LIN {X 0,Y 195.393,Z 454.313,A -85,B 0,C 180,E1 -23353.111,E2 -23353.111} C_VEL
LIN {X 0,Y 194.613,Z 444.182,A -85,B 0,C 180,E1 -23355.96,E2 -23355.96} C_VEL
LIN {X 0,Y 193.145,Z 436.002,A -85,B 0,C 180,E1 -23358.369,E2 -23358.369} C_VEL
LIN {X 0,Y 190.426,Z 427.797,A -85,B 0,C 180,E1 -23361.14,E2 -23361.14} C_VEL
LIN {X 0,Y 187.179,Z 420.29,A -85,B 0,C 180,E1 -23363.977,E2 -23363.977} C_VEL
LIN {X 0,Y 183.425,Z 413.236,A -85,B 0,C 180,E1 -23367.07,E2 -23367.07} C_VEL
LIN {X 0,Y 181.652,Z 409.98,A -85,B 0,C 180,E1 -23368.592,E2 -23368.592} C_VEL
LIN {X 0,Y 179.184,Z 405.781,A -85,B 0,C 180,E1 -23370.721,E2 -23370.721} C_VEL
LIN {X 0,Y 176.213,Z 401.753,A -85,B 0,C 180,E1 -23373.34,E2 -23373.34} C_VEL
LIN {X 0,Y 175.243,Z 399.934,A -85,B 0,C 180,E1 -23374.302,E2 -23374.302} C_VEL
LIN {X 0,Y 172.386,Z 396.823,A -85,B 0,C 180,E1 -23377.054,E2 -23377.054} C_VEL
LIN {X 0,Y 171.129,Z 394.282,A -85,B 0,C 180,E1 -23378.577,E2 -23378.577} C_VEL
LIN {X 0,Y 167.914,Z 391.613,A -85,B 0,C 180,E1 -23382.335,E2 -23382.335} C_VEL
LIN {X 0,Y 166.254,Z 388.555,A -85,B 0,C 180,E1 -23385.072,E2 -23385.072} C_VEL
LIN {X 0,Y 166.146,Z 388.15,A -85,B 0,C 180,E1 -23385.457,E2 -23385.457} C_VEL
LIN {X 0,Y 166.298,Z 387.582,A -85,B 0,C 180,E1 -23390.267,E2 -23390.267} C_VEL
LIN {X 0,Y 166.273,Z 387.45,A -85,B 0,C 180,E1 -23395.15,E2 -23395.15} C_VEL
LIN {X 0,Y 166.781,Z 387.561,A -85,B 0,C 180,E1 -23400,E2 -23400} C_VEL
LIN {X 0,Y 166.489,Z 388.269,A -85,B 0,C 180,E1 -23404.843,E2 -23404.843} C_VEL
LIN {X 0,Y 166.58,Z 389.214,A -85,B 0,C 180,E1 -23409.715,E2 -23409.715} C_VEL
LIN {X 0,Y 166.697,Z 390.162,A -85,B 0,C 180,E1 -23412.858,E2 -23412.858} C_VEL
LIN {X 0,Y 168.099,Z 393.319,A -85,B 0,C 180,E1 -23415.147,E2 -23415.147} C_VEL
LIN {X 0,Y 171.251,Z 396.71,A -85,B 0,C 180,E1 -23418.855,E2 -23418.855} C_VEL
LIN {X 0,Y 171.981,Z 397.621,A -85,B 0,C 180,E1 -23419.625,E2 -23419.625} C_VEL
LIN {X 0,Y 173.741,Z 401.026,A -85,B 0,C 180,E1 -23421.583,E2 -23421.583} C_VEL
LIN {X 0,Y 176.205,Z 403.912,A -85,B 0,C 180,E1 -23423.818,E2 -23423.818} C_VEL
LIN {X 0,Y 178.445,Z 408.052,A -85,B 0,C 180,E1 -23425.903,E2 -23425.903} C_VEL
LIN {X 0,Y 179.87,Z 410.061,A -85,B 0,C 180,E1 -23427.085,E2 -23427.085} C_VEL
LIN {X 0,Y 182.312,Z 414.458,A -85,B 0,C 180,E1 -23429.122,E2 -23429.122} C_VEL
LIN {X 0,Y 183.669,Z 417.262,A -85,B 0,C 180,E1 -23430.305,E2 -23430.305} C_VEL
LIN {X 0,Y 185.712,Z 421.013,A -85,B 0,C 180,E1 -23431.912,E2 -23431.912} C_VEL
LIN {X 0,Y 189.672,Z 429.746,A -85,B 0,C 180,E1 -23435.182,E2 -23435.182} C_VEL
LIN {X 0,Y 193.411,Z 440.1,A -85,B 0,C 180,E1 -23438.605,E2 -23438.605} C_VEL
LIN {X 0,Y 195.794,Z 448.846,A -85,B 0,C 180,E1 -23441.232,E2 -23441.232} C_VEL
LIN {X 0,Y 195.872,Z 455.455,A -85,B 0,C 180,E1 -23442.769,E2 -23442.769} C_VEL
LIN {X 0,Y 194.863,Z 467.884,A -85,B 0,C 180,E1 -23445.671,E2 -23445.671} C_VEL
LIN {X 0,Y 193.774,Z 474.064,A -85,B 0,C 180,E1 -23447.152,E2 -23447.152} C_VEL
LIN {X 0,Y 188.97,Z 484.708,A -85,B 0,C 180,E1 -23449.394,E2 -23449.394} C_VEL
LIN {X 0,Y 183.723,Z 495.484,A -85,B 0,C 180,E1 -23452.261,E2 -23452.261} C_VEL
LIN {X 0,Y 179.025,Z 504.532,A -85,B 0,C 180,E1 -23455.287,E2 -23455.287} C_VEL
LIN {X 0,Y 174.37,Z 513.451,A -85,B 0,C 180,E1 -23459.076,E2 -23459.076} C_VEL
LIN {X 0,Y 170.178,Z 520.786,A -85,B 0,C 180,E1 -23462.981,E2 -23462.981} C_VEL
LIN {X 0,Y 166.593,Z 527.552,A -85,B 0,C 180,E1 -23467.686,E2 -23467.686} C_VEL
LIN {X 0,Y 164.027,Z 532.799,A -85,B 0,C 180,E1 -23472.546,E2 -23472.546} C_VEL
LIN {X 0,Y 162.495,Z 536.663,A -85,B 0,C 180,E1 -23477.511,E2 -23477.511} C_VEL
LIN {X 0,Y 161.925,Z 539.221,A -85,B 0,C 180,E1 -23482.518,E2 -23482.518} C_VEL
LIN {X 0,Y 161.964,Z 540.31,A -85,B 0,C 180,E1 -23486.392,E2 -23486.392} C_VEL
LIN {X 0,Y 162.166,Z 540.683,A -85,B 0,C 180,E1 -23490,E2 -23490} C_VEL
LIN {X 0,Y 161.945,Z 540.01,A -85,B 0,C 180,E1 -23494.979,E2 -23494.979} C_VEL
LIN {X 0,Y 162.104,Z 538.06,A -85,B 0,C 180,E1 -23499.994,E2 -23499.994} C_VEL
LIN {X 0,Y 163.129,Z 534.845,A -85,B 0,C 180,E1 -23504.981,E2 -23504.981} C_VEL
LIN {X 0,Y 165.326,Z 529.872,A -85,B 0,C 180,E1 -23510.278,E2 -23510.278} C_VEL
LIN {X 0,Y 165.698,Z 527.731,A -85,B 0,C 180,E1 -23512.183,E2 -23512.183} C_VEL
LIN {X 0,Y 164.607,Z 520.58,A -85,B 0,C 180,E1 -23517.854,E2 -23517.854} C_VEL
LIN {X 0,Y 165.371,Z 517.795,A -85,B 0,C 180,E1 -23519.642,E2 -23519.642} C_VEL
LIN {X 0,Y 165.926,Z 516.803,A -85,B 0,C 180,E1 -23520.201,E2 -23520.201} C_VEL
LIN {X 0,Y 170.168,Z 509.415,A -85,B 0,C 180,E1 -23523.835,E2 -23523.835} C_VEL
LIN {X 0,Y 175.497,Z 499.649,A -85,B 0,C 180,E1 -23527.641,E2 -23527.641} C_VEL
LIN {X 0,Y 180.783,Z 489.726,A -85,B 0,C 180,E1 -23530.629,E2 -23530.629} C_VEL
LIN {X 0,Y 185.516,Z 480.008,A -85,B 0,C 180,E1 -23532.993,E2 -23532.993} C_VEL
LIN {X 0,Y 187.889,Z 474.908,A -85,B 0,C 180,E1 -23534.042,E2 -23534.042} C_VEL
LIN {X 0,Y 189.104,Z 468.404,A -85,B 0,C 180,E1 -23535.678,E2 -23535.678} C_VEL
LIN {X 0,Y 190.178,Z 457.705,A -85,B 0,C 180,E1 -23538.304,E2 -23538.304} C_VEL
LIN {X 0,Y 190.26,Z 451.9,A -85,B 0,C 180,E1 -23539.727,E2 -23539.727} C_VEL
LIN {X 0,Y 188.045,Z 442.99,A -85,B 0,C 180,E1 -23542.603,E2 -23542.603} C_VEL
LIN {X 0,Y 184.882,Z 433.595,A -85,B 0,C 180,E1 -23545.896,E2 -23545.896} C_VEL
LIN {X 0,Y 180.855,Z 424.352,A -85,B 0,C 180,E1 -23549.657,E2 -23549.657} C_VEL
LIN {X 0,Y 178.545,Z 419.648,A -85,B 0,C 180,E1 -23551.813,E2 -23551.813} C_VEL
LIN {X 0,Y 176.166,Z 414.939,A -85,B 0,C 180,E1 -23554.13,E2 -23554.13} C_VEL
LIN {X 0,Y 173.783,Z 410.864,A -85,B 0,C 180,E1 -23556.462,E2 -23556.462} C_VEL
LIN {X 0,Y 173.009,Z 409.372,A -85,B 0,C 180,E1 -23557.3,E2 -23557.3} C_VEL
LIN {X 0,Y 170.455,Z 405.778,A -85,B 0,C 180,E1 -23560.026,E2 -23560.026} C_VEL
LIN {X 0,Y 169.384,Z 403.444,A -85,B 0,C 180,E1 -23561.4,E2 -23561.4} C_VEL
LIN {X 0,Y 166.445,Z 399.985,A -85,B 0,C 180,E1 -23565.149,E2 -23565.149} C_VEL
LIN {X 0,Y 165.014,Z 396.727,A -85,B 0,C 180,E1 -23567.705,E2 -23567.705} C_VEL
LIN {X 0,Y 161.043,Z 391.856,A -85,B 0,C 180,E1 -23579.375,E2 -23579.375} C_VEL
LIN {X 0,Y 160.969,Z 391.971,A -85,B 0,C 180,E1 -23583.129,E2 -23583.129} C_VEL
LIN {X 0,Y 162.436,Z 393.477,A -85,B 0,C 180,E1 -23589.967,E2 -23589.967} C_VEL
LIN {X 0,Y 164.736,Z 395.178,A -85,B 0,C 180,E1 -23594.668,E2 -23594.668} C_VEL
LIN {X 0,Y 166.487,Z 398.565,A -85,B 0,C 180,E1 -23597.822,E2 -23597.822} C_VEL
LIN {X 0,Y 169.25,Z 401.27,A -85,B 0,C 180,E1 -23601.306,E2 -23601.306} C_VEL
LIN {X 0,Y 171.208,Z 404.731,A -85,B 0,C 180,E1 -23603.754,E2 -23603.754} C_VEL
LIN {X 0,Y 173.066,Z 406.867,A -85,B 0,C 180,E1 -23605.642,E2 -23605.642} C_VEL
LIN {X 0,Y 175.344,Z 410.764,A -85,B 0,C 180,E1 -23608.016,E2 -23608.016} C_VEL
LIN {X 0,Y 176.352,Z 412.26,A -85,B 0,C 180,E1 -23608.977,E2 -23608.977} C_VEL
LIN {X 0,Y 178.854,Z 416.578,A -85,B 0,C 180,E1 -23611.332,E2 -23611.332} C_VEL
LIN {X 0,Y 182.86,Z 425.001,A -85,B 0,C 180,E1 -23615.206,E2 -23615.206} C_VEL
LIN {X 0,Y 185.603,Z 431.859,A -85,B 0,C 180,E1 -23617.976,E2 -23617.976} C_VEL
LIN {X 0,Y 188.024,Z 439.877,A -85,B 0,C 180,E1 -23620.855,E2 -23620.855} C_VEL
LIN {X 0,Y 189.257,Z 448.168,A -85,B 0,C 180,E1 -23623.433,E2 -23623.433} C_VEL
LIN {X 0,Y 189.561,Z 457.642,A -85,B 0,C 180,E1 -23626.248,E2 -23626.248} C_VEL
LIN {X 0,Y 189.172,Z 465.85,A -85,B 0,C 180,E1 -23628.72,E2 -23628.72} C_VEL
LIN {X 0,Y 184.394,Z 476.022,A -85,B 0,C 180,E1 -23631.032,E2 -23631.032} C_VEL
LIN {X 0,Y 179.225,Z 486.127,A -85,B 0,C 180,E1 -23633.971,E2 -23633.971} C_VEL
LIN {X 0,Y 174.332,Z 494.554,A -85,B 0,C 180,E1 -23637.027,E2 -23637.027} C_VEL
LIN {X 0,Y 169.265,Z 502.826,A -85,B 0,C 180,E1 -23640.883,E2 -23640.883} C_VEL
LIN {X 0,Y 165.213,Z 509.295,A -85,B 0,C 180,E1 -23644.825,E2 -23644.825} C_VEL
LIN {X 0,Y 162.079,Z 513.891,A -85,B 0,C 180,E1 -23648.372,E2 -23648.372} C_VEL
LIN {X 0,Y 158.968,Z 518.703,A -85,B 0,C 180,E1 -23653.3,E2 -23653.3} C_VEL
LIN {X 0,Y 157.248,Z 521.421,A -85,B 0,C 180,E1 -23657.087,E2 -23657.087} C_VEL
LIN {X 0,Y 155.856,Z 523.863,A -85,B 0,C 180,E1 -23662.225,E2 -23662.225} C_VEL
LIN {X 0,Y 155.244,Z 525.075,A -85,B 0,C 180,E1 -23667.406,E2 -23667.406} C_VEL
LIN {X 0,Y 155.243,Z 525.092,A -85,B 0,C 180,E1 -23672.595,E2 -23672.595} C_VEL
LIN {X 0,Y 155.843,Z 523.918,A -85,B 0,C 180,E1 -23677.776,E2 -23677.776} C_VEL
LIN {X 0,Y 157.224,Z 521.516,A -85,B 0,C 180,E1 -23682.915,E2 -23682.915} C_VEL
LIN {X 0,Y 159.622,Z 517.803,A -85,B 0,C 180,E1 -23687.951,E2 -23687.951} C_VEL
LIN {X 0,Y 162.96,Z 512.68,A -85,B 0,C 180,E1 -23692.84,E2 -23692.84} C_VEL
LIN {X 0,Y 167.574,Z 505.93,A -85,B 0,C 180,E1 -23697.474,E2 -23697.474} C_VEL
LIN {X 0,Y 171.316,Z 499.691,A -85,B 0,C 180,E1 -23700.851,E2 -23700.851} C_VEL
LIN {X 0,Y 175.795,Z 492.225,A -85,B 0,C 180,E1 -23704.036,E2 -23704.036} C_VEL
LIN {X 0,Y 180.803,Z 483.334,A -85,B 0,C 180,E1 -23707.05,E2 -23707.05} C_VEL
LIN {X 0,Y 185.27,Z 474.58,A -85,B 0,C 180,E1 -23709.45,E2 -23709.45} C_VEL
LIN {X 0,Y 189.178,Z 466.217,A -85,B 0,C 180,E1 -23711.332,E2 -23711.332} C_VEL
LIN {X 0,Y 189.7,Z 457.039,A -85,B 0,C 180,E1 -23714.074,E2 -23714.074} C_VEL
LIN {X 0,Y 189.241,Z 447.251,A -85,B 0,C 180,E1 -23717.016,E2 -23717.016} C_VEL
LIN {X 0,Y 188.199,Z 440.269,A -85,B 0,C 180,E1 -23719.191,E2 -23719.191} C_VEL
LIN {X 0,Y 185.8,Z 432.24,A -85,B 0,C 180,E1 -23722.072,E2 -23722.072} C_VEL
LIN {X 0,Y 183.073,Z 425.374,A -85,B 0,C 180,E1 -23724.841,E2 -23724.841} C_VEL
LIN {X 0,Y 180.248,Z 419.479,A -85,B 0,C 180,E1 -23727.532,E2 -23727.532} C_VEL
LIN {X 0,Y 177.7,Z 414.784,A -85,B 0,C 180,E1 -23729.963,E2 -23729.963} C_VEL
LIN {X 0,Y 175.829,Z 411.344,A -85,B 0,C 180,E1 -23731.825,E2 -23731.825} C_VEL
LIN {X 0,Y 173.238,Z 407.243,A -85,B 0,C 180,E1 -23734.466,E2 -23734.466} C_VEL
LIN {X 0,Y 172.591,Z 406.168,A -85,B 0,C 180,E1 -23735.169,E2 -23735.169} C_VEL
LIN {X 0,Y 169.982,Z 402.838,A -85,B 0,C 180,E1 -23738.074,E2 -23738.074} C_VEL
LIN {X 0,Y 169.081,Z 400.884,A -85,B 0,C 180,E1 -23739.31,E2 -23739.31} C_VEL
LIN {X 0,Y 166.009,Z 397.887,A -85,B 0,C 180,E1 -23743.395,E2 -23743.395} C_VEL
LIN {X 0,Y 164.617,Z 394.969,A -85,B 0,C 180,E1 -23746.124,E2 -23746.124} C_VEL
LIN {X 0,Y 161.437,Z 392.628,A -85,B 0,C 180,E1 -23755.005,E2 -23755.005} C_VEL
LIN {X 0,Y 161.292,Z 392.143,A -85,B 0,C 180,E1 -23760.312,E2 -23760.312} C_VEL
LIN {X 0,Y 165.093,Z 396.741,A -85,B 0,C 180,E1 -23771.977,E2 -23771.977} C_VEL
LIN {X 0,Y 166.773,Z 400.471,A -85,B 0,C 180,E1 -23774.997,E2 -23774.997} C_VEL
LIN {X 0,Y 169.727,Z 403.84,A -85,B 0,C 180,E1 -23778.717,E2 -23778.717} C_VEL
LIN {X 0,Y 171.482,Z 407.457,A -85,B 0,C 180,E1 -23780.919,E2 -23780.919} C_VEL
LIN {X 0,Y 173.548,Z 410.102,A -85,B 0,C 180,E1 -23783.019,E2 -23783.019} C_VEL
LIN {X 0,Y 175.603,Z 414.134,A -85,B 0,C 180,E1 -23785.165,E2 -23785.165} C_VEL
LIN {X 0,Y 176.756,Z 415.923,A -85,B 0,C 180,E1 -23786.253,E2 -23786.253} C_VEL
LIN {X 0,Y 179.11,Z 420.459,A -85,B 0,C 180,E1 -23788.489,E2 -23788.489} C_VEL
LIN {X 0,Y 183.413,Z 429.887,A -85,B 0,C 180,E1 -23792.541,E2 -23792.541} C_VEL
LIN {X 0,Y 186.483,Z 438.016,A -85,B 0,C 180,E1 -23795.588,E2 -23795.588} C_VEL
LIN {X 0,Y 189.279,Z 447.398,A -85,B 0,C 180,E1 -23798.763,E2 -23798.763} C_VEL
LIN {X 0,Y 190.487,Z 453.178,A -85,B 0,C 180,E1 -23800.562,E2 -23800.562} C_VEL
LIN {X 0,Y 189.786,Z 463.401,A -85,B 0,C 180,E1 -23802.998,E2 -23802.998} C_VEL
LIN {X 0,Y 188.374,Z 473.627,A -85,B 0,C 180,E1 -23805.611,E2 -23805.611} C_VEL
LIN {X 0,Y 187.37,Z 476.406,A -85,B 0,C 180,E1 -23806.211,E2 -23806.211} C_VEL
LIN {X 0,Y 181.684,Z 488.144,A -85,B 0,C 180,E1 -23808.882,E2 -23808.882} C_VEL
LIN {X 0,Y 176.386,Z 498.329,A -85,B 0,C 180,E1 -23811.859,E2 -23811.859} C_VEL
LIN {X 0,Y 171.648,Z 506.944,A -85,B 0,C 180,E1 -23815.024,E2 -23815.024} C_VEL
LIN {X 0,Y 166.927,Z 515.366,A -85,B 0,C 180,E1 -23818.952,E2 -23818.952} C_VEL
LIN {X 0,Y 162.73,Z 522.284,A -85,B 0,C 180,E1 -23823.033,E2 -23823.033} C_VEL
LIN {X 0,Y 159.13,Z 528.766,A -85,B 0,C 180,E1 -23828.042,E2 -23828.042} C_VEL
LIN {X 0,Y 156.681,Z 533.558,A -85,B 0,C 180,E1 -23833.048,E2 -23833.048} C_VEL
LIN {X 0,Y 155.494,Z 536.313,A -85,B 0,C 180,E1 -23836.939,E2 -23836.939} C_VEL
LIN {X 0,Y 154.843,Z 538.873,A -85,B 0,C 180,E1 -23842.174,E2 -23842.174} C_VEL
LIN {X 0,Y 154.896,Z 540.028,A -85,B 0,C 180,E1 -23846.55,E2 -23846.55} C_VEL
LIN {X 0,Y 155.067,Z 540.337,A -85,B 0,C 180,E1 -23850,E2 -23850} C_VEL
LIN {X 0,Y 154.847,Z 539.663,A -85,B 0,C 180,E1 -23855.208,E2 -23855.208} C_VEL
LIN {X 0,Y 155.061,Z 537.716,A -85,B 0,C 180,E1 -23860.445,E2 -23860.445} C_VEL
LIN {X 0,Y 156.22,Z 534.495,A -85,B 0,C 180,E1 -23865.66,E2 -23865.66} C_VEL
LIN {X 0,Y 158.378,Z 529.931,A -85,B 0,C 180,E1 -23870.793,E2 -23870.793} C_VEL
LIN {X 0,Y 161.722,Z 523.915,A -85,B 0,C 180,E1 -23875.758,E2 -23875.758} C_VEL
LIN {X 0,Y 165.926,Z 516.803,A -85,B 0,C 180,E1 -23880.201,E2 -23880.201} C_VEL
LIN {X 0,Y 166.549,Z 514.834,A -85,B 0,C 180,E1 -23881.374,E2 -23881.374} C_VEL
LIN {X 0,Y 165.825,Z 511.72,A -85,B 0,C 180,E1 -23883.429,E2 -23883.429} C_VEL
LIN {X 0,Y 165.203,Z 508.379,A -85,B 0,C 180,E1 -23885.461,E2 -23885.461} C_VEL
LIN {X 0,Y 165.957,Z 506.053,A -85,B 0,C 180,E1 -23886.552,E2 -23886.552} C_VEL
LIN {X 0,Y 171.658,Z 496.157,A -85,B 0,C 180,E1 -23890.153,E2 -23890.153} C_VEL
LIN {X 0,Y 177.275,Z 485.624,A -85,B 0,C 180,E1 -23893.147,E2 -23893.147} C_VEL
LIN {X 0,Y 181.89,Z 476.458,A -85,B 0,C 180,E1 -23895.201,E2 -23895.201} C_VEL
LIN {X 0,Y 182.827,Z 473.07,A -85,B 0,C 180,E1 -23896.05,E2 -23896.05} C_VEL
LIN {X 0,Y 184.336,Z 462.781,A -85,B 0,C 180,E1 -23898.78,E2 -23898.78} C_VEL
LIN {X 0,Y 184.912,Z 456.848,A -85,B 0,C 180,E1 -23900.262,E2 -23900.262} C_VEL
LIN {X 0,Y 184.616,Z 454.071,A -85,B 0,C 180,E1 -23901.101,E2 -23901.101} C_VEL
LIN {X 0,Y 182.464,Z 445.092,A -85,B 0,C 180,E1 -23904.244,E2 -23904.244} C_VEL
LIN {X 0,Y 179.577,Z 436.033,A -85,B 0,C 180,E1 -23907.736,E2 -23907.736} C_VEL
LIN {X 0,Y 176.174,Z 427.807,A -85,B 0,C 180,E1 -23911.399,E2 -23911.399} C_VEL
LIN {X 0,Y 173.147,Z 421.04,A -85,B 0,C 180,E1 -23914.774,E2 -23914.774} C_VEL
LIN {X 0,Y 170.899,Z 416.946,A -85,B 0,C 180,E1 -23917.244,E2 -23917.244} C_VEL
LIN {X 0,Y 170.268,Z 415.613,A -85,B 0,C 180,E1 -23918.034,E2 -23918.034} C_VEL
LIN {X 0,Y 167.786,Z 411.62,A -85,B 0,C 180,E1 -23921.058,E2 -23921.058} C_VEL
LIN {X 0,Y 166.994,Z 409.815,A -85,B 0,C 180,E1 -23922.235,E2 -23922.235} C_VEL
LIN {X 0,Y 164.212,Z 405.951,A -85,B 0,C 180,E1 -23926.386,E2 -23926.386} C_VEL
LIN {X 0,Y 163.205,Z 403.395,A -85,B 0,C 180,E1 -23928.512,E2 -23928.512} C_VEL
LIN {X 0,Y 159.915,Z 398.72,A -85,B 0,C 180,E1 -23940,E2 -23940} C_VEL
LIN {X 0,Y 160.226,Z 399.536,A -85,B 0,C 180,E1 -23946.296,E2 -23946.296} C_VEL
LIN {X 0,Y 163.048,Z 401.904,A -85,B 0,C 180,E1 -23954.032,E2 -23954.032} C_VEL
LIN {X 0,Y 164.671,Z 405.31,A -85,B 0,C 180,E1 -23957.383,E2 -23957.383} C_VEL
LIN {X 0,Y 166.989,Z 407.8,A -85,B 0,C 180,E1 -23960.639,E2 -23960.639} C_VEL
LIN {X 0,Y 168.889,Z 411.278,A -85,B 0,C 180,E1 -23963.287,E2 -23963.287} C_VEL
LIN {X 0,Y 170.284,Z 413.024,A -85,B 0,C 180,E1 -23964.879,E2 -23964.879} C_VEL
LIN {X 0,Y 171.813,Z 416.056,A -85,B 0,C 180,E1 -23966.741,E2 -23966.741} C_VEL
LIN {X 0,Y 172.951,Z 417.649,A -85,B 0,C 180,E1 -23967.936,E2 -23967.936} C_VEL
LIN {X 0,Y 176.446,Z 424.882,A -85,B 0,C 180,E1 -23971.855,E2 -23971.855} C_VEL
LIN {X 0,Y 179.315,Z 431.782,A -85,B 0,C 180,E1 -23975.086,E2 -23975.086} C_VEL
LIN {X 0,Y 181.477,Z 437.95,A -85,B 0,C 180,E1 -23977.689,E2 -23977.689} C_VEL
LIN {X 0,Y 183.036,Z 444.155,A -85,B 0,C 180,E1 -23980.027,E2 -23980.027} C_VEL
LIN {X 0,Y 183.88,Z 452.358,A -85,B 0,C 180,E1 -23982.725,E2 -23982.725} C_VEL
LIN {X 0,Y 183.857,Z 460.777,A -85,B 0,C 180,E1 -23985.373,E2 -23985.373} C_VEL
LIN {X 0,Y 183.416,Z 467.29,A -85,B 0,C 180,E1 -23987.482,E2 -23987.482} C_VEL
LIN {X 0,Y 178.018,Z 478.189,A -85,B 0,C 180,E1 -23990.093,E2 -23990.093} C_VEL
LIN {X 0,Y 172.671,Z 487.974,A -85,B 0,C 180,E1 -23993.105,E2 -23993.105} C_VEL
LIN {X 0,Y 166.851,Z 497.382,A -85,B 0,C 180,E1 -23996.799,E2 -23996.799} C_VEL
LIN {X 0,Y 162.071,Z 504.783,A -85,B 0,C 180,E1 -24000.612,E2 -24000.612} C_VEL
LIN {X 0,Y 157.645,Z 511.263,A -85,B 0,C 180,E1 -24004.943,E2 -24004.943} C_VEL
LIN {X 0,Y 153.708,Z 516.83,A -85,B 0,C 180,E1 -24009.945,E2 -24009.945} C_VEL
LIN {X 0,Y 151.502,Z 520.061,A -85,B 0,C 180,E1 -24013.839,E2 -24013.839} C_VEL
LIN {X 0,Y 149.468,Z 523.144,A -85,B 0,C 180,E1 -24019.159,E2 -24019.159} C_VEL
LIN {X 0,Y 148.385,Z 524.966,A -85,B 0,C 180,E1 -24024.565,E2 -24024.565} C_VEL
LIN {X 0,Y 148.085,Z 525.577,A -85,B 0,C 180,E1 -24030,E2 -24030} C_VEL
LIN {X 0,Y 148.385,Z 525.001,A -85,B 0,C 180,E1 -24035.436,E2 -24035.436} C_VEL
LIN {X 0,Y 149.45,Z 523.219,A -85,B 0,C 180,E1 -24040.842,E2 -24040.842} C_VEL
LIN {X 0,Y 151.465,Z 520.173,A -85,B 0,C 180,E1 -24046.165,E2 -24046.165} C_VEL
LIN {X 0,Y 154.499,Z 515.775,A -85,B 0,C 180,E1 -24051.341,E2 -24051.341} C_VEL
LIN {X 0,Y 158.783,Z 509.873,A -85,B 0,C 180,E1 -24056.271,E2 -24056.271} C_VEL
LIN {X 0,Y 162.567,Z 504.115,A -85,B 0,C 180,E1 -24059.958,E2 -24059.958} C_VEL
LIN {X 0,Y 167.524,Z 496.479,A -85,B 0,C 180,E1 -24063.771,E2 -24063.771} C_VEL
LIN {X 0,Y 172.615,Z 488.342,A -85,B 0,C 180,E1 -24066.91,E2 -24066.91} C_VEL
LIN {X 0,Y 177.926,Z 478.632,A -85,B 0,C 180,E1 -24069.932,E2 -24069.932} C_VEL
LIN {X 0,Y 182.91,Z 468.797,A -85,B 0,C 180,E1 -24072.318,E2 -24072.318} C_VEL
LIN {X 0,Y 183.566,Z 466.653,A -85,B 0,C 180,E1 -24072.892,E2 -24072.892} C_VEL
LIN {X 0,Y 184.057,Z 457.45,A -85,B 0,C 180,E1 -24075.826,E2 -24075.826} C_VEL
LIN {X 0,Y 183.728,Z 448.637,A -85,B 0,C 180,E1 -24078.65,E2 -24078.65} C_VEL
LIN {X 0,Y 182.849,Z 442.842,A -85,B 0,C 180,E1 -24080.638,E2 -24080.638} C_VEL
LIN {X 0,Y 180.741,Z 435.478,A -85,B 0,C 180,E1 -24083.54,E2 -24083.54} C_VEL
LIN {X 0,Y 178.209,Z 428.792,A -85,B 0,C 180,E1 -24086.487,E2 -24086.487} C_VEL
LIN {X 0,Y 175.157,Z 421.928,A -85,B 0,C 180,E1 -24089.897,E2 -24089.897} C_VEL
LIN {X 0,Y 173.111,Z 417.951,A -85,B 0,C 180,E1 -24092.168,E2 -24092.168} C_VEL
LIN {X 0,Y 170.339,Z 413.123,A -85,B 0,C 180,E1 -24095.375,E2 -24095.375} C_VEL
LIN {X 0,Y 167.411,Z 408.739,A -85,B 0,C 180,E1 -24099.094,E2 -24099.094} C_VEL
LIN {X 0,Y 166.845,Z 407.464,A -85,B 0,C 180,E1 -24099.986,E2 -24099.986} C_VEL
LIN {X 0,Y 164.018,Z 404.24,A -85,B 0,C 180,E1 -24104.306,E2 -24104.306} C_VEL
LIN {X 0,Y 163.037,Z 401.815,A -85,B 0,C 180,E1 -24106.602,E2 -24106.602} C_VEL
LIN {X 0,Y 160.286,Z 399.656,A -85,B 0,C 180,E1 -24114.969,E2 -24114.969} C_VEL
LIN {X 0,Y 160.167,Z 399.081,A -85,B 0,C 180,E1 -24120,E2 -24120} C_VEL
LIN {X 0,Y 163.29,Z 403.434,A -85,B 0,C 180,E1 -24131.167,E2 -24131.167} C_VEL
LIN {X 0,Y 165.384,Z 407.876,A -85,B 0,C 180,E1 -24135.244,E2 -24135.244} C_VEL
LIN {X 0,Y 167.415,Z 410.422,A -85,B 0,C 180,E1 -24138.035,E2 -24138.035} C_VEL
LIN {X 0,Y 169.322,Z 414.314,A -85,B 0,C 180,E1 -24140.659,E2 -24140.659} C_VEL
LIN {X 0,Y 170.8,Z 416.547,A -85,B 0,C 180,E1 -24142.371,E2 -24142.371} C_VEL
LIN {X 0,Y 172.204,Z 419.621,A -85,B 0,C 180,E1 -24144.086,E2 -24144.086} C_VEL
LIN {X 0,Y 173.325,Z 421.24,A -85,B 0,C 180,E1 -24145.198,E2 -24145.198} C_VEL
LIN {X 0,Y 177.362,Z 430.35,A -85,B 0,C 180,E1 -24149.689,E2 -24149.689} C_VEL
LIN {X 0,Y 180.392,Z 438.258,A -85,B 0,C 180,E1 -24153.054,E2 -24153.054} C_VEL
LIN {X 0,Y 183.162,Z 447.385,A -85,B 0,C 180,E1 -24156.492,E2 -24156.492} C_VEL
LIN {X 0,Y 185.013,Z 455.771,A -85,B 0,C 180,E1 -24159.375,E2 -24159.375} C_VEL
LIN {X 0,Y 184.495,Z 462.871,A -85,B 0,C 180,E1 -24161.197,E2 -24161.197} C_VEL
LIN {X 0,Y 182.654,Z 474.627,A -85,B 0,C 180,E1 -24164.308,E2 -24164.308} C_VEL
LIN {X 0,Y 181.21,Z 478.249,A -85,B 0,C 180,E1 -24165.14,E2 -24165.14} C_VEL
LIN {X 0,Y 175.408,Z 489.554,A -85,B 0,C 180,E1 -24167.846,E2 -24167.846} C_VEL
LIN {X 0,Y 169.932,Z 499.459,A -85,B 0,C 180,E1 -24170.897,E2 -24170.897} C_VEL
LIN {X 0,Y 165.072,Z 507.844,A -85,B 0,C 180,E1 -24174.159,E2 -24174.159} C_VEL
LIN {X 0,Y 160.148,Z 516.067,A -85,B 0,C 180,E1 -24178.222,E2 -24178.222} C_VEL
LIN {X 0,Y 156.349,Z 521.927,A -85,B 0,C 180,E1 -24181.836,E2 -24181.836} C_VEL
LIN {X 0,Y 153.379,Z 526.848,A -85,B 0,C 180,E1 -24185.644,E2 -24185.644} C_VEL
LIN {X 0,Y 150.38,Z 532.099,A -85,B 0,C 180,E1 -24190.904,E2 -24190.904} C_VEL
LIN {X 0,Y 148.512,Z 535.965,A -85,B 0,C 180,E1 -24196.313,E2 -24196.313} C_VEL
LIN {X 0,Y 147.765,Z 538.526,A -85,B 0,C 180,E1 -24201.796,E2 -24201.796} C_VEL
LIN {X 0,Y 147.823,Z 539.823,A -85,B 0,C 180,E1 -24207.275,E2 -24207.275} C_VEL
LIN {X 0,Y 147.97,Z 539.992,A -85,B 0,C 180,E1 -24210,E2 -24210} C_VEL
LIN {X 0,Y 147.817,Z 539.745,A -85,B 0,C 180,E1 -24213.2,E2 -24213.2} C_VEL
LIN {X 0,Y 147.772,Z 538.498,A -85,B 0,C 180,E1 -24218.203,E2 -24218.203} C_VEL
LIN {X 0,Y 148.509,Z 535.916,A -85,B 0,C 180,E1 -24223.687,E2 -24223.687} C_VEL
LIN {X 0,Y 150.346,Z 532.034,A -85,B 0,C 180,E1 -24229.1,E2 -24229.1} C_VEL
LIN {X 0,Y 153.349,Z 526.76,A -85,B 0,C 180,E1 -24234.36,E2 -24234.36} C_VEL
LIN {X 0,Y 157.485,Z 519.957,A -85,B 0,C 180,E1 -24239.399,E2 -24239.399} C_VEL
LIN {X 0,Y 162.136,Z 512.58,A -85,B 0,C 180,E1 -24243.55,E2 -24243.55} C_VEL
LIN {X 0,Y 165.957,Z 506.053,A -85,B 0,C 180,E1 -24246.552,E2 -24246.552} C_VEL
LIN {X 0,Y 167.514,Z 502.526,A -85,B 0,C 180,E1 -24248.075,E2 -24248.075} C_VEL
LIN {X 0,Y 169.57,Z 491.512,A -85,B 0,C 180,E1 -24252.826,E2 -24252.826} C_VEL
LIN {X 0,Y 170.994,Z 487.438,A -85,B 0,C 180,E1 -24254.187,E2 -24254.187} C_VEL
LIN {X 0,Y 171.692,Z 486.011,A -85,B 0,C 180,E1 -24254.577,E2 -24254.577} C_VEL
LIN {X 0,Y 176.534,Z 476.683,A -85,B 0,C 180,E1 -24256.728,E2 -24256.728} C_VEL
LIN {X 0,Y 178.317,Z 468.131,A -85,B 0,C 180,E1 -24259.115,E2 -24259.115} C_VEL
LIN {X 0,Y 179.433,Z 459.049,A -85,B 0,C 180,E1 -24261.569,E2 -24261.569} C_VEL
LIN {X 0,Y 178.035,Z 451.308,A -85,B 0,C 180,E1 -24264.391,E2 -24264.391} C_VEL
LIN {X 0,Y 175.698,Z 442.476,A -85,B 0,C 180,E1 -24267.927,E2 -24267.927} C_VEL
LIN {X 0,Y 172.888,Z 434.648,A -85,B 0,C 180,E1 -24271.516,E2 -24271.516} C_VEL
LIN {X 0,Y 169.614,Z 426.604,A -85,B 0,C 180,E1 -24275.724,E2 -24275.724} C_VEL
LIN {X 0,Y 167.096,Z 421.434,A -85,B 0,C 180,E1 -24279.053,E2 -24279.053} C_VEL
LIN {X 0,Y 164.861,Z 417.041,A -85,B 0,C 180,E1 -24282.318,E2 -24282.318} C_VEL
LIN {X 0,Y 164.084,Z 415.744,A -85,B 0,C 180,E1 -24283.516,E2 -24283.516} C_VEL
LIN {X 0,Y 161.773,Z 411.615,A -85,B 0,C 180,E1 -24287.773,E2 -24287.773} C_VEL
LIN {X 0,Y 161.314,Z 410.138,A -85,B 0,C 180,E1 -24289.012,E2 -24289.012} C_VEL
LIN {X 0,Y 158.513,Z 405.698,A -85,B 0,C 180,E1 -24300,E2 -24300} C_VEL
LIN {X 0,Y 158.776,Z 406.508,A -85,B 0,C 180,E1 -24306.354,E2 -24306.354} C_VEL
LIN {X 0,Y 161.165,Z 408.719,A -85,B 0,C 180,E1 -24313.556,E2 -24313.556} C_VEL
LIN {X 0,Y 162.686,Z 412.09,A -85,B 0,C 180,E1 -24317.116,E2 -24317.116} C_VEL
LIN {X 0,Y 164.551,Z 414.354,A -85,B 0,C 180,E1 -24320.061,E2 -24320.061} C_VEL
LIN {X 0,Y 166.012,Z 417.291,A -85,B 0,C 180,E1 -24322.397,E2 -24322.397} C_VEL
LIN {X 0,Y 167.242,Z 418.892,A -85,B 0,C 180,E1 -24323.986,E2 -24323.986} C_VEL
LIN {X 0,Y 169.992,Z 424.516,A -85,B 0,C 180,E1 -24327.718,E2 -24327.718} C_VEL
LIN {X 0,Y 172.846,Z 430.879,A -85,B 0,C 180,E1 -24331.365,E2 -24331.365} C_VEL
LIN {X 0,Y 175.546,Z 438.377,A -85,B 0,C 180,E1 -24335.013,E2 -24335.013} C_VEL
LIN {X 0,Y 177.359,Z 445.118,A -85,B 0,C 180,E1 -24337.893,E2 -24337.893} C_VEL
LIN {X 0,Y 178.24,Z 450.556,A -85,B 0,C 180,E1 -24339.968,E2 -24339.968} C_VEL
LIN {X 0,Y 178.455,Z 458.836,A -85,B 0,C 180,E1 -24342.793,E2 -24342.793} C_VEL
LIN {X 0,Y 177.66,Z 468.822,A -85,B 0,C 180,E1 -24346.168,E2 -24346.168} C_VEL
LIN {X 0,Y 172.629,Z 478.581,A -85,B 0,C 180,E1 -24348.581,E2 -24348.581} C_VEL
LIN {X 0,Y 167.061,Z 488.349,A -85,B 0,C 180,E1 -24351.647,E2 -24351.647} C_VEL
LIN {X 0,Y 161.774,Z 496.533,A -85,B 0,C 180,E1 -24354.857,E2 -24354.857} C_VEL
LIN {X 0,Y 156.493,Z 504.241,A -85,B 0,C 180,E1 -24358.772,E2 -24358.772} C_VEL
LIN {X 0,Y 152.485,Z 510.004,A -85,B 0,C 180,E1 -24362.555,E2 -24362.555} C_VEL
LIN {X 0,Y 147.954,Z 515.969,A -85,B 0,C 180,E1 -24367.666,E2 -24367.666} C_VEL
LIN {X 0,Y 144.694,Z 520.408,A -85,B 0,C 180,E1 -24373.057,E2 -24373.057} C_VEL
LIN {X 0,Y 142.494,Z 523.491,A -85,B 0,C 180,E1 -24378.622,E2 -24378.622} C_VEL
LIN {X 0,Y 141.331,Z 525.311,A -85,B 0,C 180,E1 -24384.292,E2 -24384.292} C_VEL
LIN {X 0,Y 140.994,Z 525.923,A -85,B 0,C 180,E1 -24390,E2 -24390} C_VEL
LIN {X 0,Y 141.331,Z 525.345,A -85,B 0,C 180,E1 -24395.708,E2 -24395.708} C_VEL
LIN {X 0,Y 142.479,Z 523.564,A -85,B 0,C 180,E1 -24401.38,E2 -24401.38} C_VEL
LIN {X 0,Y 144.663,Z 520.518,A -85,B 0,C 180,E1 -24406.948,E2 -24406.948} C_VEL
LIN {X 0,Y 147.89,Z 516.122,A -85,B 0,C 180,E1 -24412.345,E2 -24412.345} C_VEL
LIN {X 0,Y 152.457,Z 510.223,A -85,B 0,C 180,E1 -24417.451,E2 -24417.451} C_VEL
LIN {X 0,Y 157.044,Z 503.637,A -85,B 0,C 180,E1 -24421.757,E2 -24421.757} C_VEL
LIN {X 0,Y 162.496,Z 495.619,A -85,B 0,C 180,E1 -24425.724,E2 -24425.724} C_VEL
LIN {X 0,Y 167.883,Z 487.245,A -85,B 0,C 180,E1 -24428.899,E2 -24428.899} C_VEL
LIN {X 0,Y 173.566,Z 477.248,A -85,B 0,C 180,E1 -24431.922,E2 -24431.922} C_VEL
LIN {X 0,Y 177.705,Z 469.135,A -85,B 0,C 180,E1 -24433.893,E2 -24433.893} C_VEL
LIN {X 0,Y 178.398,Z 462.294,A -85,B 0,C 180,E1 -24436.206,E2 -24436.206} C_VEL
LIN {X 0,Y 178.548,Z 454.097,A -85,B 0,C 180,E1 -24438.993,E2 -24438.993} C_VEL
LIN {X 0,Y 177.992,Z 447.743,A -85,B 0,C 180,E1 -24441.26,E2 -24441.26} C_VEL
LIN {X 0,Y 176.373,Z 440.844,A -85,B 0,C 180,E1 -24444.097,E2 -24444.097} C_VEL
LIN {X 0,Y 173.83,Z 433.366,A -85,B 0,C 180,E1 -24447.608,E2 -24447.608} C_VEL
LIN {X 0,Y 171.605,Z 427.737,A -85,B 0,C 180,E1 -24450.563,E2 -24450.563} C_VEL
LIN {X 0,Y 169.095,Z 422.681,A -85,B 0,C 180,E1 -24453.775,E2 -24453.775} C_VEL
LIN {X 0,Y 167.162,Z 418.774,A -85,B 0,C 180,E1 -24456.458,E2 -24456.458} C_VEL
LIN {X 0,Y 164.725,Z 414.722,A -85,B 0,C 180,E1 -24460.042,E2 -24460.042} C_VEL
LIN {X 0,Y 164.179,Z 413.758,A -85,B 0,C 180,E1 -24460.949,E2 -24460.949} C_VEL
LIN {X 0,Y 161.84,Z 410.515,A -85,B 0,C 180,E1 -24465.218,E2 -24465.218} C_VEL
LIN {X 0,Y 161.028,Z 408.516,A -85,B 0,C 180,E1 -24467.395,E2 -24467.395} C_VEL
LIN {X 0,Y 158.83,Z 406.622,A -85,B 0,C 180,E1 -24474.922,E2 -24474.922} C_VEL
LIN {X 0,Y 158.734,Z 406.114,A -85,B 0,C 180,E1 -24480,E2 -24480} C_VEL
LIN {X 0,Y 161.479,Z 410.251,A -85,B 0,C 180,E1 -24490.818,E2 -24490.818} C_VEL
LIN {X 0,Y 162.921,Z 413.957,A -85,B 0,C 180,E1 -24494.202,E2 -24494.202} C_VEL
LIN {X 0,Y 164.893,Z 416.843,A -85,B 0,C 180,E1 -24497.358,E2 -24497.358} C_VEL
LIN {X 0,Y 166.391,Z 420.247,A -85,B 0,C 180,E1 -24499.749,E2 -24499.749} C_VEL
LIN {X 0,Y 167.292,Z 421.616,A -85,B 0,C 180,E1 -24500.921,E2 -24500.921} C_VEL
LIN {X 0,Y 170.054,Z 427.478,A -85,B 0,C 180,E1 -24504.601,E2 -24504.601} C_VEL
LIN {X 0,Y 173.541,Z 436.1,A -85,B 0,C 180,E1 -24509.076,E2 -24509.076} C_VEL
LIN {X 0,Y 176.268,Z 444.238,A -85,B 0,C 180,E1 -24512.701,E2 -24512.701} C_VEL
LIN {X 0,Y 178.491,Z 453.139,A -85,B 0,C 180,E1 -24516.2,E2 -24516.2} C_VEL
LIN {X 0,Y 179.573,Z 459.441,A -85,B 0,C 180,E1 -24518.486,E2 -24518.486} C_VEL
LIN {X 0,Y 178.388,Z 468.403,A -85,B 0,C 180,E1 -24520.89,E2 -24520.89} C_VEL
LIN {X 0,Y 176.675,Z 476.875,A -85,B 0,C 180,E1 -24523.287,E2 -24523.287} C_VEL
LIN {X 0,Y 171.147,Z 487.363,A -85,B 0,C 180,E1 -24525.725,E2 -24525.725} C_VEL
LIN {X 0,Y 165.349,Z 497.579,A -85,B 0,C 180,E1 -24528.79,E2 -24528.79} C_VEL
LIN {X 0,Y 159.465,Z 507.168,A -85,B 0,C 180,E1 -24532.495,E2 -24532.495} C_VEL
LIN {X 0,Y 154.063,Z 515.708,A -85,B 0,C 180,E1 -24536.81,E2 -24536.81} C_VEL
LIN {X 0,Y 150.04,Z 521.57,A -85,B 0,C 180,E1 -24540.538,E2 -24540.538} C_VEL
LIN {X 0,Y 145.852,Z 528.108,A -85,B 0,C 180,E1 -24545.972,E2 -24545.972} C_VEL
LIN {X 0,Y 143.014,Z 532.857,A -85,B 0,C 180,E1 -24551.372,E2 -24551.372} C_VEL
LIN {X 0,Y 141.552,Z 535.616,A -85,B 0,C 180,E1 -24555.626,E2 -24555.626} C_VEL
LIN {X 0,Y 140.685,Z 538.178,A -85,B 0,C 180,E1 -24561.38,E2 -24561.38} C_VEL
LIN {X 0,Y 140.734,Z 539.477,A -85,B 0,C 180,E1 -24567.137,E2 -24567.137} C_VEL
LIN {X 0,Y 140.877,Z 539.646,A -85,B 0,C 180,E1 -24570,E2 -24570} C_VEL
LIN {X 0,Y 140.734,Z 539.471,A -85,B 0,C 180,E1 -24572.862,E2 -24572.862} C_VEL
LIN {X 0,Y 140.717,Z 538.151,A -85,B 0,C 180,E1 -24578.617,E2 -24578.617} C_VEL
LIN {X 0,Y 141.548,Z 535.567,A -85,B 0,C 180,E1 -24584.374,E2 -24584.374} C_VEL
LIN {X 0,Y 143.583,Z 531.683,A -85,B 0,C 180,E1 -24590.037,E2 -24590.037} C_VEL
LIN {X 0,Y 146.816,Z 526.405,A -85,B 0,C 180,E1 -24595.52,E2 -24595.52} C_VEL
LIN {X 0,Y 151.269,Z 519.599,A -85,B 0,C 180,E1 -24600.735,E2 -24600.735} C_VEL
LIN {X 0,Y 156.157,Z 512.213,A -85,B 0,C 180,E1 -24605.018,E2 -24605.018} C_VEL
LIN {X 0,Y 161.713,Z 503.278,A -85,B 0,C 180,E1 -24609.062,E2 -24609.062} C_VEL
LIN {X 0,Y 167.203,Z 494.125,A -85,B 0,C 180,E1 -24612.262,E2 -24612.262} C_VEL
LIN {X 0,Y 171.692,Z 486.011,A -85,B 0,C 180,E1 -24614.577,E2 -24614.577} C_VEL
LIN {X 0,Y 173.317,Z 481.752,A -85,B 0,C 180,E1 -24615.816,E2 -24615.816} C_VEL
LIN {X 0,Y 173.919,Z 477.636,A -85,B 0,C 180,E1 -24617.223,E2 -24617.223} C_VEL
LIN {X 0,Y 173.714,Z 469.588,A -85,B 0,C 180,E1 -24620.232,E2 -24620.232} C_VEL
LIN {X 0,Y 173.827,Z 463.885,A -85,B 0,C 180,E1 -24622.16,E2 -24622.16} C_VEL
LIN {X 0,Y 174.014,Z 462.06,A -85,B 0,C 180,E1 -24622.713,E2 -24622.713} C_VEL
LIN {X 0,Y 172.679,Z 454.024,A -85,B 0,C 180,E1 -24625.885,E2 -24625.885} C_VEL
LIN {X 0,Y 170.859,Z 446.313,A -85,B 0,C 180,E1 -24629.196,E2 -24629.196} C_VEL
LIN {X 0,Y 168.56,Z 439.196,A -85,B 0,C 180,E1 -24632.701,E2 -24632.701} C_VEL
LIN {X 0,Y 166.273,Z 432.732,A -85,B 0,C 180,E1 -24636.249,E2 -24636.249} C_VEL
LIN {X 0,Y 163.897,Z 427.274,A -85,B 0,C 180,E1 -24639.938,E2 -24639.938} C_VEL
LIN {X 0,Y 161.801,Z 422.555,A -85,B 0,C 180,E1 -24643.601,E2 -24643.601} C_VEL
LIN {X 0,Y 159.463,Z 418.117,A -85,B 0,C 180,E1 -24648.4,E2 -24648.4} C_VEL
LIN {X 0,Y 159.016,Z 416.645,A -85,B 0,C 180,E1 -24649.818,E2 -24649.818} C_VEL
LIN {X 0,Y 156.795,Z 412.654,A -85,B 0,C 180,E1 -24660,E2 -24660} C_VEL
LIN {X 0,Y 156.787,Z 413.044,A -85,B 0,C 180,E1 -24664.5,E2 -24664.5} C_VEL
LIN {X 0,Y 158.921,Z 415.178,A -85,B 0,C 180,E1 -24672.775,E2 -24672.775} C_VEL
LIN {X 0,Y 159.739,Z 417.567,A -85,B 0,C 180,E1 -24675.307,E2 -24675.307} C_VEL
LIN {X 0,Y 161.754,Z 420.339,A -85,B 0,C 180,E1 -24679.164,E2 -24679.164} C_VEL
LIN {X 0,Y 164.492,Z 425.978,A -85,B 0,C 180,E1 -24683.948,E2 -24683.948} C_VEL
LIN {X 0,Y 166.475,Z 430.309,A -85,B 0,C 180,E1 -24686.99,E2 -24686.99} C_VEL
LIN {X 0,Y 168.9,Z 436.374,A -85,B 0,C 180,E1 -24690.654,E2 -24690.654} C_VEL
LIN {X 0,Y 171.49,Z 444.967,A -85,B 0,C 180,E1 -24695.012,E2 -24695.012} C_VEL
LIN {X 0,Y 172.85,Z 451.991,A -85,B 0,C 180,E1 -24698.088,E2 -24698.088} C_VEL
LIN {X 0,Y 173.047,Z 459.596,A -85,B 0,C 180,E1 -24700.912,E2 -24700.912} C_VEL
LIN {X 0,Y 172.18,Z 469.105,A -85,B 0,C 180,E1 -24704.321,E2 -24704.321} C_VEL
LIN {X 0,Y 171.975,Z 470.404,A -85,B 0,C 180,E1 -24704.778,E2 -24704.778} C_VEL
LIN {X 0,Y 168.428,Z 477.204,A -85,B 0,C 180,E1 -24706.489,E2 -24706.489} C_VEL
LIN {X 0,Y 162.492,Z 487.257,A -85,B 0,C 180,E1 -24709.551,E2 -24709.551} C_VEL
LIN {X 0,Y 156.883,Z 495.663,A -85,B 0,C 180,E1 -24712.788,E2 -24712.788} C_VEL
LIN {X 0,Y 151.154,Z 503.685,A -85,B 0,C 180,E1 -24716.818,E2 -24716.818} C_VEL
LIN {X 0,Y 146.227,Z 510.358,A -85,B 0,C 180,E1 -24721.274,E2 -24721.274} C_VEL
LIN {X 0,Y 141.396,Z 516.319,A -85,B 0,C 180,E1 -24726.57,E2 -24726.57} C_VEL
LIN {X 0,Y 137.922,Z 520.754,A -85,B 0,C 180,E1 -24732.198,E2 -24732.198} C_VEL
LIN {X 0,Y 135.552,Z 523.836,A -85,B 0,C 180,E1 -24738.031,E2 -24738.031} C_VEL
LIN {X 0,Y 134.271,Z 525.657,A -85,B 0,C 180,E1 -24743.991,E2 -24743.991} C_VEL
LIN {X 0,Y 133.905,Z 526.268,A -85,B 0,C 180,E1 -24750,E2 -24750} C_VEL
LIN {X 0,Y 134.271,Z 525.69,A -85,B 0,C 180,E1 -24756.009,E2 -24756.009} C_VEL
LIN {X 0,Y 135.54,Z 523.909,A -85,B 0,C 180,E1 -24761.971,E2 -24761.971} C_VEL
LIN {X 0,Y 137.894,Z 520.862,A -85,B 0,C 180,E1 -24767.807,E2 -24767.807} C_VEL
LIN {X 0,Y 141.334,Z 516.468,A -85,B 0,C 180,E1 -24773.442,E2 -24773.442} C_VEL
LIN {X 0,Y 146.201,Z 510.573,A -85,B 0,C 180,E1 -24778.732,E2 -24778.732} C_VEL
LIN {X 0,Y 150.847,Z 504.267,A -85,B 0,C 180,E1 -24783.004,E2 -24783.004} C_VEL
LIN {X 0,Y 156.785,Z 495.981,A -85,B 0,C 180,E1 -24787.24,E2 -24787.24} C_VEL
LIN {X 0,Y 162.411,Z 487.616,A -85,B 0,C 180,E1 -24790.474,E2 -24790.474} C_VEL
LIN {X 0,Y 168.358,Z 477.634,A -85,B 0,C 180,E1 -24793.535,E2 -24793.535} C_VEL
LIN {X 0,Y 172.08,Z 470.669,A -85,B 0,C 180,E1 -24795.282,E2 -24795.282} C_VEL
LIN {X 0,Y 172.992,Z 462.642,A -85,B 0,C 180,E1 -24798.156,E2 -24798.156} C_VEL
LIN {X 0,Y 173.123,Z 454.001,A -85,B 0,C 180,E1 -24801.324,E2 -24801.324} C_VEL
LIN {X 0,Y 172.311,Z 448.18,A -85,B 0,C 180,E1 -24803.744,E2 -24803.744} C_VEL
LIN {X 0,Y 170.217,Z 440.197,A -85,B 0,C 180,E1 -24807.537,E2 -24807.537} C_VEL
LIN {X 0,Y 167.881,Z 433.497,A -85,B 0,C 180,E1 -24811.222,E2 -24811.222} C_VEL
LIN {X 0,Y 166.329,Z 429.633,A -85,B 0,C 180,E1 -24813.662,E2 -24813.662} C_VEL
LIN {X 0,Y 163.994,Z 424.729,A -85,B 0,C 180,E1 -24817.312,E2 -24817.312} C_VEL
LIN {X 0,Y 161.882,Z 420.648,A -85,B 0,C 180,E1 -24820.997,E2 -24820.997} C_VEL
LIN {X 0,Y 159.388,Z 416.538,A -85,B 0,C 180,E1 -24826.317,E2 -24826.317} C_VEL
LIN {X 0,Y 158.922,Z 415.205,A -85,B 0,C 180,E1 -24827.874,E2 -24827.874} C_VEL
LIN {X 0,Y 157.074,Z 413.513,A -85,B 0,C 180,E1 -24834.865,E2 -24834.865} C_VEL
LIN {X 0,Y 157.006,Z 413.026,A -85,B 0,C 180,E1 -24840,E2 -24840} C_VEL
LIN {X 0,Y 159.273,Z 416.914,A -85,B 0,C 180,E1 -24850.246,E2 -24850.246} C_VEL
LIN {X 0,Y 160.632,Z 420.693,A -85,B 0,C 180,E1 -24853.924,E2 -24853.924} C_VEL
LIN {X 0,Y 162.023,Z 422.71,A -85,B 0,C 180,E1 -24856.376,E2 -24856.376} C_VEL
LIN {X 0,Y 163.103,Z 425.736,A -85,B 0,C 180,E1 -24858.562,E2 -24858.562} C_VEL
LIN {X 0,Y 164.085,Z 427.485,A -85,B 0,C 180,E1 -24860.038,E2 -24860.038} C_VEL
LIN {X 0,Y 166.712,Z 433.929,A -85,B 0,C 180,E1 -24864.219,E2 -24864.219} C_VEL
LIN {X 0,Y 169.541,Z 441.748,A -85,B 0,C 180,E1 -24868.47,E2 -24868.47} C_VEL
LIN {X 0,Y 171.79,Z 449.591,A -85,B 0,C 180,E1 -24872.129,E2 -24872.129} C_VEL
LIN {X 0,Y 173.37,Z 457.171,A -85,B 0,C 180,E1 -24875.294,E2 -24875.294} C_VEL
LIN {X 0,Y 174.123,Z 462.22,A -85,B 0,C 180,E1 -24877.26,E2 -24877.26} C_VEL
LIN {X 0,Y 173.237,Z 468.173,A -85,B 0,C 180,E1 -24878.972,E2 -24878.972} C_VEL
LIN {X 0,Y 171.085,Z 477.869,A -85,B 0,C 180,E1 -24881.842,E2 -24881.842} C_VEL
LIN {X 0,Y 165.054,Z 488.773,A -85,B 0,C 180,E1 -24884.502,E2 -24884.502} C_VEL
LIN {X 0,Y 159.043,Z 498.707,A -85,B 0,C 180,E1 -24887.631,E2 -24887.631} C_VEL
LIN {X 0,Y 153.344,Z 507.488,A -85,B 0,C 180,E1 -24891.181,E2 -24891.181} C_VEL
LIN {X 0,Y 148.107,Z 515.35,A -85,B 0,C 180,E1 -24895.289,E2 -24895.289} C_VEL
LIN {X 0,Y 143.831,Z 521.215,A -85,B 0,C 180,E1 -24899.131,E2 -24899.131} C_VEL
LIN {X 0,Y 139.405,Z 527.61,A -85,B 0,C 180,E1 -24904.627,E2 -24904.627} C_VEL
LIN {X 0,Y 136.227,Z 532.506,A -85,B 0,C 180,E1 -24910.406,E2 -24910.406} C_VEL
LIN {X 0,Y 134.613,Z 535.267,A -85,B 0,C 180,E1 -24914.867,E2 -24914.867} C_VEL
LIN {X 0,Y 133.632,Z 537.831,A -85,B 0,C 180,E1 -24920.922,E2 -24920.922} C_VEL
LIN {X 0,Y 133.634,Z 539.132,A -85,B 0,C 180,E1 -24926.985,E2 -24926.985} C_VEL
LIN {X 0,Y 133.785,Z 539.301,A -85,B 0,C 180,E1 -24930,E2 -24930} C_VEL
LIN {X 0,Y 133.634,Z 539.125,A -85,B 0,C 180,E1 -24933.014,E2 -24933.014} C_VEL
LIN {X 0,Y 133.657,Z 537.803,A -85,B 0,C 180,E1 -24939.076,E2 -24939.076} C_VEL
LIN {X 0,Y 134.607,Z 535.217,A -85,B 0,C 180,E1 -24945.133,E2 -24945.133} C_VEL
LIN {X 0,Y 136.858,Z 531.332,A -85,B 0,C 180,E1 -24951.067,E2 -24951.067} C_VEL
LIN {X 0,Y 140.357,Z 526.05,A -85,B 0,C 180,E1 -24956.785,E2 -24956.785} C_VEL
LIN {X 0,Y 145.142,Z 519.24,A -85,B 0,C 180,E1 -24962.184,E2 -24962.184} C_VEL
LIN {X 0,Y 150.322,Z 511.848,A -85,B 0,C 180,E1 -24966.591,E2 -24966.591} C_VEL
LIN {X 0,Y 156.195,Z 502.903,A -85,B 0,C 180,E1 -24970.725,E2 -24970.725} C_VEL
LIN {X 0,Y 161.969,Z 493.737,A -85,B 0,C 180,E1 -24973.968,E2 -24973.968} C_VEL
LIN {X 0,Y 167.123,Z 484.813,A -85,B 0,C 180,E1 -24976.503,E2 -24976.503} C_VEL
LIN {X 0,Y 170.991,Z 477.635,A -85,B 0,C 180,E1 -24978.173,E2 -24978.173} C_VEL
LIN {X 0,Y 173.158,Z 467.943,A -85,B 0,C 180,E1 -24981.02,E2 -24981.02} C_VEL
LIN {X 0,Y 173.827,Z 463.885,A -85,B 0,C 180,E1 -24982.16,E2 -24982.16} C_VEL
LIN {X 0,Y 173.713,Z 461.255,A -85,B 0,C 180,E1 -24983.104,E2 -24983.104} C_VEL
LIN {X 0,Y 172.99,Z 459.07,A -85,B 0,C 180,E1 -24984.148,E2 -24984.148} C_VEL
LIN {X 0,Y 170.514,Z 455.661,A -85,B 0,C 180,E1 -24986.397,E2 -24986.397} C_VEL
LIN {X 0,Y 166.465,Z 450.898,A -85,B 0,C 180,E1 -24990.028,E2 -24990.028} C_VEL
LIN {X 0,Y 165.664,Z 448.82,A -85,B 0,C 180,E1 -24991.215,E2 -24991.215} C_VEL
LIN {X 0,Y 163.514,Z 441.467,A -85,B 0,C 180,E1 -24995.225,E2 -24995.225} C_VEL
LIN {X 0,Y 162.52,Z 438.267,A -85,B 0,C 180,E1 -24997.096,E2 -24997.096} C_VEL
LIN {X 0,Y 160.499,Z 433.024,A -85,B 0,C 180,E1 -25000.828,E2 -25000.828} C_VEL
LIN {X 0,Y 158.705,Z 428.532,A -85,B 0,C 180,E1 -25004.592,E2 -25004.592} C_VEL
LIN {X 0,Y 156.766,Z 423.821,A -85,B 0,C 180,E1 -25009.67,E2 -25009.67} C_VEL
LIN {X 0,Y 155.233,Z 421.39,A -85,B 0,C 180,E1 -25014.805,E2 -25014.805} C_VEL
LIN {X 0,Y 154.781,Z 419.501,A -85,B 0,C 180,E1 -25020,E2 -25020} C_VEL
LIN {X 0,Y 154.705,Z 419.53,A -85,B 0,C 180,E1 -25022.604,E2 -25022.604} C_VEL
LIN {X 0,Y 155.841,Z 421.261,A -85,B 0,C 180,E1 -25030.393,E2 -25030.393} C_VEL
LIN {X 0,Y 156.671,Z 422.385,A -85,B 0,C 180,E1 -25032.962,E2 -25032.962} C_VEL
LIN {X 0,Y 157.45,Z 424.58,A -85,B 0,C 180,E1 -25035.535,E2 -25035.535} C_VEL
LIN {X 0,Y 158.598,Z 426.358,A -85,B 0,C 180,E1 -25038.071,E2 -25038.071} C_VEL
LIN {X 0,Y 161.086,Z 431.74,A -85,B 0,C 180,E1 -25043.121,E2 -25043.121} C_VEL
LIN {X 0,Y 162.465,Z 434.973,A -85,B 0,C 180,E1 -25045.632,E2 -25045.632} C_VEL
LIN {X 0,Y 164.486,Z 440.897,A -85,B 0,C 180,E1 -25049.431,E2 -25049.431} C_VEL
LIN {X 0,Y 166.397,Z 447.962,A -85,B 0,C 180,E1 -25053.304,E2 -25053.304} C_VEL
LIN {X 0,Y 167.653,Z 454.996,A -85,B 0,C 180,E1 -25056.681,E2 -25056.681} C_VEL
LIN {X 0,Y 167.76,Z 460.499,A -85,B 0,C 180,E1 -25058.932,E2 -25058.932} C_VEL
LIN {X 0,Y 167.068,Z 467.628,A -85,B 0,C 180,E1 -25061.648,E2 -25061.648} C_VEL
LIN {X 0,Y 166.424,Z 471.95,A -85,B 0,C 180,E1 -25063.295,E2 -25063.295} C_VEL
LIN {X 0,Y 163.353,Z 477.596,A -85,B 0,C 180,E1 -25064.774,E2 -25064.774} C_VEL
LIN {X 0,Y 157.156,Z 487.632,A -85,B 0,C 180,E1 -25067.871,E2 -25067.871} C_VEL
LIN {X 0,Y 151.301,Z 496.031,A -85,B 0,C 180,E1 -25071.165,E2 -25071.165} C_VEL
LIN {X 0,Y 144.983,Z 504.393,A -85,B 0,C 180,E1 -25075.495,E2 -25075.495} C_VEL
LIN {X 0,Y 140.049,Z 510.711,A -85,B 0,C 180,E1 -25079.879,E2 -25079.879} C_VEL
LIN {X 0,Y 134.898,Z 516.668,A -85,B 0,C 180,E1 -25085.368,E2 -25085.368} C_VEL
LIN {X 0,Y 131.173,Z 521.1,A -85,B 0,C 180,E1 -25091.248,E2 -25091.248} C_VEL
LIN {X 0,Y 128.602,Z 524.182,A -85,B 0,C 180,E1 -25097.374,E2 -25097.374} C_VEL
LIN {X 0,Y 127.224,Z 526.002,A -85,B 0,C 180,E1 -25103.657,E2 -25103.657} C_VEL
LIN {X 0,Y 126.818,Z 526.613,A -85,B 0,C 180,E1 -25110,E2 -25110} C_VEL
LIN {X 0,Y 127.224,Z 526.035,A -85,B 0,C 180,E1 -25116.343,E2 -25116.343} C_VEL
LIN {X 0,Y 128.59,Z 524.254,A -85,B 0,C 180,E1 -25122.628,E2 -25122.628} C_VEL
LIN {X 0,Y 131.132,Z 521.208,A -85,B 0,C 180,E1 -25128.758,E2 -25128.758} C_VEL
LIN {X 0,Y 134.838,Z 516.815,A -85,B 0,C 180,E1 -25134.644,E2 -25134.644} C_VEL
LIN {X 0,Y 140.026,Z 510.922,A -85,B 0,C 180,E1 -25140.127,E2 -25140.127} C_VEL
LIN {X 0,Y 144.704,Z 504.918,A -85,B 0,C 180,E1 -25144.344,E2 -25144.344} C_VEL
LIN {X 0,Y 151.2,Z 496.342,A -85,B 0,C 180,E1 -25148.867,E2 -25148.867} C_VEL
LIN {X 0,Y 157.087,Z 487.986,A -85,B 0,C 180,E1 -25152.152,E2 -25152.152} C_VEL
LIN {X 0,Y 163.301,Z 478.019,A -85,B 0,C 180,E1 -25155.245,E2 -25155.245} C_VEL
LIN {X 0,Y 165.536,Z 474.219,A -85,B 0,C 180,E1 -25156.2,E2 -25156.2} C_VEL
LIN {X 0,Y 166.492,Z 472.236,A -85,B 0,C 180,E1 -25156.761,E2 -25156.761} C_VEL
LIN {X 0,Y 167.544,Z 464.694,A -85,B 0,C 180,E1 -25159.628,E2 -25159.628} C_VEL
LIN {X 0,Y 167.885,Z 458.801,A -85,B 0,C 180,E1 -25161.91,E2 -25161.91} C_VEL
LIN {X 0,Y 167.577,Z 453.828,A -85,B 0,C 180,E1 -25164.045,E2 -25164.045} C_VEL
LIN {X 0,Y 166.299,Z 447.143,A -85,B 0,C 180,E1 -25167.324,E2 -25167.324} C_VEL
LIN {X 0,Y 164.33,Z 440.295,A -85,B 0,C 180,E1 -25171.203,E2 -25171.203} C_VEL
LIN {X 0,Y 162.663,Z 435.34,A -85,B 0,C 180,E1 -25174.401,E2 -25174.401} C_VEL
LIN {X 0,Y 160.661,Z 430.592,A -85,B 0,C 180,E1 -25178.171,E2 -25178.171} C_VEL
LIN {X 0,Y 158.815,Z 426.692,A -85,B 0,C 180,E1 -25181.954,E2 -25181.954} C_VEL
LIN {X 0,Y 156.855,Z 422.85,A -85,B 0,C 180,E1 -25187.054,E2 -25187.054} C_VEL
LIN {X 0,Y 156.11,Z 421.452,A -85,B 0,C 180,E1 -25189.625,E2 -25189.625} C_VEL
LIN {X 0,Y 154.9,Z 419.912,A -85,B 0,C 180,E1 -25197.399,E2 -25197.399} C_VEL
LIN {X 0,Y 154.979,Z 419.858,A -85,B 0,C 180,E1 -25200,E2 -25200} C_VEL
LIN {X 0,Y 156.747,Z 423.31,A -85,B 0,C 180,E1 -25209.454,E2 -25209.454} C_VEL
LIN {X 0,Y 158.277,Z 427.729,A -85,B 0,C 180,E1 -25214.135,E2 -25214.135} C_VEL
LIN {X 0,Y 158.917,Z 428.702,A -85,B 0,C 180,E1 -25215.387,E2 -25215.387} C_VEL
LIN {X 0,Y 161.321,Z 434.963,A -85,B 0,C 180,E1 -25220.397,E2 -25220.397} C_VEL
LIN {X 0,Y 162.967,Z 439.624,A -85,B 0,C 180,E1 -25223.51,E2 -25223.51} C_VEL
LIN {X 0,Y 165.346,Z 447.282,A -85,B 0,C 180,E1 -25227.875,E2 -25227.875} C_VEL
LIN {X 0,Y 167.208,Z 455.101,A -85,B 0,C 180,E1 -25231.694,E2 -25231.694} C_VEL
LIN {X 0,Y 168.402,Z 462.673,A -85,B 0,C 180,E1 -25235.017,E2 -25235.017} C_VEL
LIN {X 0,Y 168.671,Z 465.419,A -85,B 0,C 180,E1 -25236.168,E2 -25236.168} C_VEL
LIN {X 0,Y 166.994,Z 473.668,A -85,B 0,C 180,E1 -25238.666,E2 -25238.666} C_VEL
LIN {X 0,Y 165.24,Z 479.702,A -85,B 0,C 180,E1 -25240.512,E2 -25240.512} C_VEL
LIN {X 0,Y 159.036,Z 490.182,A -85,B 0,C 180,E1 -25243.183,E2 -25243.183} C_VEL
LIN {X 0,Y 152.821,Z 499.836,A -85,B 0,C 180,E1 -25246.383,E2 -25246.383} C_VEL
LIN {X 0,Y 146.77,Z 508.652,A -85,B 0,C 180,E1 -25250.182,E2 -25250.182} C_VEL
LIN {X 0,Y 141.485,Z 516.023,A -85,B 0,C 180,E1 -25254.291,E2 -25254.291} C_VEL
LIN {X 0,Y 136.382,Z 522.6,A -85,B 0,C 180,E1 -25258.981,E2 -25258.981} C_VEL
LIN {X 0,Y 131.816,Z 528.798,A -85,B 0,C 180,E1 -25265.01,E2 -25265.01} C_VEL
LIN {X 0,Y 128.833,Z 533.154,A -85,B 0,C 180,E1 -25270.894,E2 -25270.894} C_VEL
LIN {X 0,Y 126.974,Z 536.36,A -85,B 0,C 180,E1 -25277.208,E2 -25277.208} C_VEL
LIN {X 0,Y 126.443,Z 538.292,A -85,B 0,C 180,E1 -25283.617,E2 -25283.617} C_VEL
LIN {X 0,Y 126.586,Z 538.85,A -85,B 0,C 180,E1 -25287.928,E2 -25287.928} C_VEL
LIN {X 0,Y 126.687,Z 538.955,A -85,B 0,C 180,E1 -25290,E2 -25290} C_VEL
LIN {X 0,Y 126.545,Z 538.779,A -85,B 0,C 180,E1 -25293.183,E2 -25293.183} C_VEL
LIN {X 0,Y 126.594,Z 537.454,A -85,B 0,C 180,E1 -25299.587,E2 -25299.587} C_VEL
LIN {X 0,Y 127.692,Z 534.866,A -85,B 0,C 180,E1 -25305.973,E2 -25305.973} C_VEL
LIN {X 0,Y 130.184,Z 530.98,A -85,B 0,C 180,E1 -25312.203,E2 -25312.203} C_VEL
LIN {X 0,Y 133.983,Z 525.696,A -85,B 0,C 180,E1 -25318.17,E2 -25318.17} C_VEL
LIN {X 0,Y 139.121,Z 518.883,A -85,B 0,C 180,E1 -25323.758,E2 -25323.758} C_VEL
LIN {X 0,Y 144.612,Z 511.483,A -85,B 0,C 180,E1 -25328.29,E2 -25328.29} C_VEL
LIN {X 0,Y 150.824,Z 502.53,A -85,B 0,C 180,E1 -25332.506,E2 -25332.506} C_VEL
LIN {X 0,Y 156.902,Z 493.351,A -85,B 0,C 180,E1 -25335.781,E2 -25335.781} C_VEL
LIN {X 0,Y 162.301,Z 484.409,A -85,B 0,C 180,E1 -25338.328,E2 -25338.328} C_VEL
LIN {X 0,Y 165.627,Z 478.326,A -85,B 0,C 180,E1 -25339.799,E2 -25339.799} C_VEL
LIN {X 0,Y 168.28,Z 467.223,A -85,B 0,C 180,E1 -25343.201,E2 -25343.201} C_VEL
LIN {X 0,Y 168.452,Z 464.168,A -85,B 0,C 180,E1 -25344.261,E2 -25344.261} C_VEL
LIN {X 0,Y 167.379,Z 456.48,A -85,B 0,C 180,E1 -25347.561,E2 -25347.561} C_VEL
LIN {X 0,Y 165.664,Z 448.82,A -85,B 0,C 180,E1 -25351.215,E2 -25351.215} C_VEL
LIN {X 0,Y 164.43,Z 446.077,A -85,B 0,C 180,E1 -25352.976,E2 -25352.976} C_VEL
LIN {X 0,Y 162.646,Z 444.223,A -85,B 0,C 180,E1 -25354.855,E2 -25354.855} C_VEL
LIN {X 0,Y 157.779,Z 440.392,A -85,B 0,C 180,E1 -25360.172,E2 -25360.172} C_VEL
LIN {X 0,Y 157.03,Z 438.957,A -85,B 0,C 180,E1 -25361.513,E2 -25361.513} C_VEL
LIN {X 0,Y 155.444,Z 434.389,A -85,B 0,C 180,E1 -25365.602,E2 -25365.602} C_VEL
LIN {X 0,Y 154.16,Z 430.97,A -85,B 0,C 180,E1 -25369.493,E2 -25369.493} C_VEL
LIN {X 0,Y 153.474,Z 429.232,A -85,B 0,C 180,E1 -25372.104,E2 -25372.104} C_VEL
LIN {X 0,Y 152.464,Z 426.266,A -85,B 0,C 180,E1 -25380,E2 -25380} C_VEL
LIN {X 0,Y 152.392,Z 426.261,A -85,B 0,C 180,E1 -25382.644,E2 -25382.644} C_VEL
LIN {X 0,Y 152.837,Z 427.244,A -85,B 0,C 180,E1 -25387.93,E2 -25387.93} C_VEL
LIN {X 0,Y 153.429,Z 428.036,A -85,B 0,C 180,E1 -25390.558,E2 -25390.558} C_VEL
LIN {X 0,Y 154.111,Z 429.435,A -85,B 0,C 180,E1 -25393.181,E2 -25393.181} C_VEL
LIN {X 0,Y 155.864,Z 433.432,A -85,B 0,C 180,E1 -25398.4,E2 -25398.4} C_VEL
LIN {X 0,Y 157.52,Z 437.425,A -85,B 0,C 180,E1 -25402.287,E2 -25402.287} C_VEL
LIN {X 0,Y 159.186,Z 442.541,A -85,B 0,C 180,E1 -25406.2,E2 -25406.2} C_VEL
LIN {X 0,Y 160.332,Z 446.424,A -85,B 0,C 180,E1 -25408.828,E2 -25408.828} C_VEL
LIN {X 0,Y 161.849,Z 453.46,A -85,B 0,C 180,E1 -25412.893,E2 -25412.893} C_VEL
LIN {X 0,Y 162.514,Z 459.036,A -85,B 0,C 180,E1 -25415.718,E2 -25415.718} C_VEL
LIN {X 0,Y 162.293,Z 464.809,A -85,B 0,C 180,E1 -25418.208,E2 -25418.208} C_VEL
LIN {X 0,Y 161.338,Z 471.253,A -85,B 0,C 180,E1 -25420.8,E2 -25420.8} C_VEL
LIN {X 0,Y 160.686,Z 474.167,A -85,B 0,C 180,E1 -25421.966,E2 -25421.966} C_VEL
LIN {X 0,Y 154.064,Z 484.838,A -85,B 0,C 180,E1 -25425.003,E2 -25425.003} C_VEL
LIN {X 0,Y 147.857,Z 493.726,A -85,B 0,C 180,E1 -25428.283,E2 -25428.283} C_VEL
LIN {X 0,Y 141.182,Z 502.302,A -85,B 0,C 180,E1 -25432.425,E2 -25432.425} C_VEL
LIN {X 0,Y 135.467,Z 509.289,A -85,B 0,C 180,E1 -25436.993,E2 -25436.993} C_VEL
LIN {X 0,Y 129.726,Z 515.642,A -85,B 0,C 180,E1 -25442.581,E2 -25442.581} C_VEL
LIN {X 0,Y 125.356,Z 520.442,A -85,B 0,C 180,E1 -25448.628,E2 -25448.628} C_VEL
LIN {X 0,Y 122.893,Z 523.15,A -85,B 0,C 180,E1 -25453.385,E2 -25453.385} C_VEL
LIN {X 0,Y 120.783,Z 525.591,A -85,B 0,C 180,E1 -25459.947,E2 -25459.947} C_VEL
LIN {X 0,Y 119.841,Z 526.802,A -85,B 0,C 180,E1 -25466.638,E2 -25466.638} C_VEL
LIN {X 0,Y 119.821,Z 526.818,A -85,B 0,C 180,E1 -25473.363,E2 -25473.363} C_VEL
LIN {X 0,Y 120.781,Z 525.642,A -85,B 0,C 180,E1 -25480.054,E2 -25480.054} C_VEL
LIN {X 0,Y 122.876,Z 523.239,A -85,B 0,C 180,E1 -25486.618,E2 -25486.618} C_VEL
LIN {X 0,Y 126.299,Z 519.53,A -85,B 0,C 180,E1 -25492.925,E2 -25492.925} C_VEL
LIN {X 0,Y 129.666,Z 515.808,A -85,B 0,C 180,E1 -25497.433,E2 -25497.433} C_VEL
LIN {X 0,Y 135.442,Z 509.506,A -85,B 0,C 180,E1 -25503.014,E2 -25503.014} C_VEL
LIN {X 0,Y 140.223,Z 503.671,A -85,B 0,C 180,E1 -25506.974,E2 -25506.974} C_VEL
LIN {X 0,Y 146.753,Z 495.386,A -85,B 0,C 180,E1 -25511.185,E2 -25511.185} C_VEL
LIN {X 0,Y 152.926,Z 486.834,A -85,B 0,C 180,E1 -25514.495,E2 -25514.495} C_VEL
LIN {X 0,Y 158.404,Z 478.403,A -85,B 0,C 180,E1 -25517.061,E2 -25517.061} C_VEL
LIN {X 0,Y 160.658,Z 474.619,A -85,B 0,C 180,E1 -25518.046,E2 -25518.046} C_VEL
LIN {X 0,Y 161.667,Z 470.287,A -85,B 0,C 180,E1 -25519.741,E2 -25519.741} C_VEL
LIN {X 0,Y 162.564,Z 462.941,A -85,B 0,C 180,E1 -25522.752,E2 -25522.752} C_VEL
LIN {X 0,Y 162.634,Z 459.396,A -85,B 0,C 180,E1 -25524.312,E2 -25524.312} C_VEL
LIN {X 0,Y 161.773,Z 452.597,A -85,B 0,C 180,E1 -25527.8,E2 -25527.8} C_VEL
LIN {X 0,Y 160.217,Z 445.756,A -85,B 0,C 180,E1 -25531.864,E2 -25531.864} C_VEL
LIN {X 0,Y 158.774,Z 440.8,A -85,B 0,C 180,E1 -25535.272,E2 -25535.272} C_VEL
LIN {X 0,Y 157.138,Z 436.346,A -85,B 0,C 180,E1 -25539.034,E2 -25539.034} C_VEL
LIN {X 0,Y 156.059,Z 433.788,A -85,B 0,C 180,E1 -25541.624,E2 -25541.624} C_VEL
LIN {X 0,Y 154.285,Z 429.875,A -85,B 0,C 180,E1 -25546.834,E2 -25546.834} C_VEL
LIN {X 0,Y 153.669,Z 428.285,A -85,B 0,C 180,E1 -25549.459,E2 -25549.459} C_VEL
LIN {X 0,Y 152.682,Z 427.009,A -85,B 0,C 180,E1 -25554.717,E2 -25554.717} C_VEL
LIN {X 0,Y 152.652,Z 426.603,A -85,B 0,C 180,E1 -25560,E2 -25560} C_VEL
LIN {X 0,Y 153.725,Z 429.353,A -85,B 0,C 180,E1 -25567.883,E2 -25567.883} C_VEL
LIN {X 0,Y 155.642,Z 434.592,A -85,B 0,C 180,E1 -25574.38,E2 -25574.38} C_VEL
LIN {X 0,Y 157.679,Z 440.545,A -85,B 0,C 180,E1 -25579.529,E2 -25579.529} C_VEL
LIN {X 0,Y 159.302,Z 446.175,A -85,B 0,C 180,E1 -25583.394,E2 -25583.394} C_VEL
LIN {X 0,Y 160.761,Z 451.764,A -85,B 0,C 180,E1 -25586.758,E2 -25586.758} C_VEL
LIN {X 0,Y 162.17,Z 458.933,A -85,B 0,C 180,E1 -25590.521,E2 -25590.521} C_VEL
LIN {X 0,Y 163.083,Z 466.494,A -85,B 0,C 180,E1 -25594.071,E2 -25594.071} C_VEL
LIN {X 0,Y 163.221,Z 468.855,A -85,B 0,C 180,E1 -25595.103,E2 -25595.103} C_VEL
LIN {X 0,Y 160.416,Z 479.266,A -85,B 0,C 180,E1 -25598.452,E2 -25598.452} C_VEL
LIN {X 0,Y 160.064,Z 480.342,A -85,B 0,C 180,E1 -25598.797,E2 -25598.797} C_VEL
LIN {X 0,Y 153.119,Z 491.546,A -85,B 0,C 180,E1 -25601.766,E2 -25601.766} C_VEL
LIN {X 0,Y 146.683,Z 500.96,A -85,B 0,C 180,E1 -25605.031,E2 -25605.031} C_VEL
LIN {X 0,Y 139.987,Z 510.139,A -85,B 0,C 180,E1 -25609.257,E2 -25609.257} C_VEL
LIN {X 0,Y 134.898,Z 516.693,A -85,B 0,C 180,E1 -25613.191,E2 -25613.191} C_VEL
LIN {X 0,Y 130.27,Z 522.246,A -85,B 0,C 180,E1 -25617.35,E2 -25617.35} C_VEL
LIN {X 0,Y 125.496,Z 528.251,A -85,B 0,C 180,E1 -25623.383,E2 -25623.383} C_VEL
LIN {X 0,Y 122.079,Z 532.805,A -85,B 0,C 180,E1 -25629.792,E2 -25629.792} C_VEL
LIN {X 0,Y 120.003,Z 536.013,A -85,B 0,C 180,E1 -25636.452,E2 -25636.452} C_VEL
LIN {X 0,Y 119.357,Z 537.945,A -85,B 0,C 180,E1 -25643.236,E2 -25643.236} C_VEL
LIN {X 0,Y 119.526,Z 538.533,A -85,B 0,C 180,E1 -25648.317,E2 -25648.317} C_VEL
LIN {X 0,Y 119.517,Z 538.535,A -85,B 0,C 180,E1 -25651.516,E2 -25651.516} C_VEL
LIN {X 0,Y 119.364,Z 537.927,A -85,B 0,C 180,E1 -25656.762,E2 -25656.762} C_VEL
LIN {X 0,Y 120.007,Z 535.97,A -85,B 0,C 180,E1 -25663.547,E2 -25663.547} C_VEL
LIN {X 0,Y 122.032,Z 532.742,A -85,B 0,C 180,E1 -25670.215,E2 -25670.215} C_VEL
LIN {X 0,Y 125.422,Z 528.166,A -85,B 0,C 180,E1 -25676.633,E2 -25676.633} C_VEL
LIN {X 0,Y 130.264,Z 522.134,A -85,B 0,C 180,E1 -25682.651,E2 -25682.651} C_VEL
LIN {X 0,Y 136.512,Z 514.49,A -85,B 0,C 180,E1 -25688.155,E2 -25688.155} C_VEL
LIN {X 0,Y 142.864,Z 505.986,A -85,B 0,C 180,E1 -25692.745,E2 -25692.745} C_VEL
LIN {X 0,Y 149.802,Z 496.242,A -85,B 0,C 180,E1 -25696.651,E2 -25696.651} C_VEL
LIN {X 0,Y 156.457,Z 485.943,A -85,B 0,C 180,E1 -25699.786,E2 -25699.786} C_VEL
LIN {X 0,Y 160.004,Z 480.061,A -85,B 0,C 180,E1 -25701.228,E2 -25701.228} C_VEL
LIN {X 0,Y 162.755,Z 470.212,A -85,B 0,C 180,E1 -25704.386,E2 -25704.386} C_VEL
LIN {X 0,Y 163.123,Z 468.522,A -85,B 0,C 180,E1 -25704.945,E2 -25704.945} C_VEL
LIN {X 0,Y 162.322,Z 460.276,A -85,B 0,C 180,E1 -25708.698,E2 -25708.698} C_VEL
LIN {X 0,Y 160.856,Z 452.484,A -85,B 0,C 180,E1 -25712.693,E2 -25712.693} C_VEL
LIN {X 0,Y 159.152,Z 445.946,A -85,B 0,C 180,E1 -25716.583,E2 -25716.583} C_VEL
LIN {X 0,Y 158.119,Z 442.371,A -85,B 0,C 180,E1 -25718.971,E2 -25718.971} C_VEL
LIN {X 0,Y 157.03,Z 438.957,A -85,B 0,C 180,E1 -25721.513,E2 -25721.513} C_VEL
LIN {X 0,Y 155.909,Z 437.195,A -85,B 0,C 180,E1 -25723.531,E2 -25723.531} C_VEL
LIN {X 0,Y 154.469,Z 436.437,A -85,B 0,C 180,E1 -25725.639,E2 -25725.639} C_VEL
LIN {X 0,Y 150.921,Z 435.987,A -85,B 0,C 180,E1 -25731.533,E2 -25731.533} C_VEL
LIN {X 0,Y 150.459,Z 435.499,A -85,B 0,C 180,E1 -25733.045,E2 -25733.045} C_VEL
LIN {X 0,Y 149.852,Z 432.917,A -85,B 0,C 180,E1 -25740,E2 -25740} C_VEL
LIN {X 0,Y 149.788,Z 432.877,A -85,B 0,C 180,E1 -25742.69,E2 -25742.69} C_VEL
LIN {X 0,Y 150.176,Z 433.877,A -85,B 0,C 180,E1 -25748.071,E2 -25748.071} C_VEL
LIN {X 0,Y 151.001,Z 435.504,A -85,B 0,C 180,E1 -25752.203,E2 -25752.203} C_VEL
LIN {X 0,Y 152.411,Z 439.177,A -85,B 0,C 180,E1 -25757.442,E2 -25757.442} C_VEL
LIN {X 0,Y 153.757,Z 443.023,A -85,B 0,C 180,E1 -25761.449,E2 -25761.449} C_VEL
LIN {X 0,Y 155.054,Z 447.82,A -85,B 0,C 180,E1 -25765.362,E2 -25765.362} C_VEL
LIN {X 0,Y 156.139,Z 452.548,A -85,B 0,C 180,E1 -25768.676,E2 -25768.676} C_VEL
LIN {X 0,Y 157.081,Z 458.851,A -85,B 0,C 180,E1 -25772.473,E2 -25772.473} C_VEL
LIN {X 0,Y 157.352,Z 463.161,A -85,B 0,C 180,E1 -25774.782,E2 -25774.782} C_VEL
LIN {X 0,Y 156.862,Z 468.48,A -85,B 0,C 180,E1 -25777.217,E2 -25777.217} C_VEL
LIN {X 0,Y 155.613,Z 474.607,A -85,B 0,C 180,E1 -25779.845,E2 -25779.845} C_VEL
LIN {X 0,Y 154.888,Z 476.503,A -85,B 0,C 180,E1 -25780.533,E2 -25780.533} C_VEL
LIN {X 0,Y 148.025,Z 486.832,A -85,B 0,C 180,E1 -25783.61,E2 -25783.61} C_VEL
LIN {X 0,Y 141.572,Z 495.433,A -85,B 0,C 180,E1 -25786.954,E2 -25786.954} C_VEL
LIN {X 0,Y 134.679,Z 503.762,A -85,B 0,C 180,E1 -25791.23,E2 -25791.23} C_VEL
LIN {X 0,Y 129.558,Z 509.643,A -85,B 0,C 180,E1 -25795.279,E2 -25795.279} C_VEL
LIN {X 0,Y 123.459,Z 515.991,A -85,B 0,C 180,E1 -25801.062,E2 -25801.062} C_VEL
LIN {X 0,Y 118.763,Z 520.79,A -85,B 0,C 180,E1 -25807.378,E2 -25807.378} C_VEL
LIN {X 0,Y 116.104,Z 523.496,A -85,B 0,C 180,E1 -25812.383,E2 -25812.383} C_VEL
LIN {X 0,Y 113.817,Z 525.936,A -85,B 0,C 180,E1 -25819.325,E2 -25819.325} C_VEL
LIN {X 0,Y 112.777,Z 527.146,A -85,B 0,C 180,E1 -25826.427,E2 -25826.427} C_VEL
LIN {X 0,Y 112.757,Z 527.162,A -85,B 0,C 180,E1 -25833.574,E2 -25833.574} C_VEL
LIN {X 0,Y 113.815,Z 525.986,A -85,B 0,C 180,E1 -25840.676,E2 -25840.676} C_VEL
LIN {X 0,Y 116.088,Z 523.584,A -85,B 0,C 180,E1 -25847.62,E2 -25847.62} C_VEL
LIN {X 0,Y 119.773,Z 519.876,A -85,B 0,C 180,E1 -25854.252,E2 -25854.252} C_VEL
LIN {X 0,Y 123.408,Z 516.156,A -85,B 0,C 180,E1 -25858.952,E2 -25858.952} C_VEL
LIN {X 0,Y 129.529,Z 509.858,A -85,B 0,C 180,E1 -25864.731,E2 -25864.731} C_VEL
LIN {X 0,Y 135.542,Z 502.929,A -85,B 0,C 180,E1 -25869.434,E2 -25869.434} C_VEL
LIN {X 0,Y 142.565,Z 494.41,A -85,B 0,C 180,E1 -25873.643,E2 -25873.643} C_VEL
LIN {X 0,Y 149.042,Z 485.601,A -85,B 0,C 180,E1 -25876.962,E2 -25876.962} C_VEL
LIN {X 0,Y 154.857,Z 476.951,A -85,B 0,C 180,E1 -25879.481,E2 -25879.481} C_VEL
LIN {X 0,Y 155.677,Z 475.043,A -85,B 0,C 180,E1 -25880.128,E2 -25880.128} C_VEL
LIN {X 0,Y 157.193,Z 467.107,A -85,B 0,C 180,E1 -25883.589,E2 -25883.589} C_VEL
LIN {X 0,Y 157.414,Z 461.946,A -85,B 0,C 180,E1 -25886.076,E2 -25886.076} C_VEL
LIN {X 0,Y 156.918,Z 456.721,A -85,B 0,C 180,E1 -25888.997,E2 -25888.997} C_VEL
LIN {X 0,Y 155.76,Z 450.194,A -85,B 0,C 180,E1 -25893.178,E2 -25893.178} C_VEL
LIN {X 0,Y 154.364,Z 444.942,A -85,B 0,C 180,E1 -25897.232,E2 -25897.232} C_VEL
LIN {X 0,Y 152.969,Z 440.785,A -85,B 0,C 180,E1 -25901.239,E2 -25901.239} C_VEL
LIN {X 0,Y 152.141,Z 438.6,A -85,B 0,C 180,E1 -25903.908,E2 -25903.908} C_VEL
LIN {X 0,Y 150.916,Z 435.034,A -85,B 0,C 180,E1 -25909.264,E2 -25909.264} C_VEL
LIN {X 0,Y 150.049,Z 433.606,A -85,B 0,C 180,E1 -25914.624,E2 -25914.624} C_VEL
LIN {X 0,Y 149.96,Z 433.234,A -85,B 0,C 180,E1 -25917.313,E2 -25917.313} C_VEL
LIN {X 0,Y 150.032,Z 433.244,A -85,B 0,C 180,E1 -25920,E2 -25920} C_VEL
LIN {X 0,Y 150.941,Z 436.167,A -85,B 0,C 180,E1 -25928.029,E2 -25928.029} C_VEL
LIN {X 0,Y 152.206,Z 440.338,A -85,B 0,C 180,E1 -25933.348,E2 -25933.348} C_VEL
LIN {X 0,Y 153.857,Z 446.015,A -85,B 0,C 180,E1 -25938.647,E2 -25938.647} C_VEL
LIN {X 0,Y 155.398,Z 452.518,A -85,B 0,C 180,E1 -25943.311,E2 -25943.311} C_VEL
LIN {X 0,Y 156.659,Z 459.214,A -85,B 0,C 180,E1 -25947.376,E2 -25947.376} C_VEL
LIN {X 0,Y 157.425,Z 465.425,A -85,B 0,C 180,E1 -25950.705,E2 -25950.705} C_VEL
LIN {X 0,Y 157.796,Z 471.735,A -85,B 0,C 180,E1 -25953.815,E2 -25953.815} C_VEL
LIN {X 0,Y 154.919,Z 480.97,A -85,B 0,C 180,E1 -25956.939,E2 -25956.939} C_VEL
LIN {X 0,Y 148.429,Z 491.164,A -85,B 0,C 180,E1 -25959.697,E2 -25959.697} C_VEL
LIN {X 0,Y 141.689,Z 500.586,A -85,B 0,C 180,E1 -25962.977,E2 -25962.977} C_VEL
LIN {X 0,Y 134.612,Z 509.776,A -85,B 0,C 180,E1 -25967.255,E2 -25967.255} C_VEL
LIN {X 0,Y 129.222,Z 516.334,A -85,B 0,C 180,E1 -25971.284,E2 -25971.284} C_VEL
LIN {X 0,Y 124.289,Z 521.893,A -85,B 0,C 180,E1 -25975.565,E2 -25975.565} C_VEL
LIN {X 0,Y 119.109,Z 527.9,A -85,B 0,C 180,E1 -25981.833,E2 -25981.833} C_VEL
LIN {X 0,Y 115.345,Z 532.455,A -85,B 0,C 180,E1 -25988.556,E2 -25988.556} C_VEL
LIN {X 0,Y 113.045,Z 535.665,A -85,B 0,C 180,E1 -25995.6,E2 -25995.6} C_VEL
LIN {X 0,Y 112.265,Z 537.597,A -85,B 0,C 180,E1 -26002.807,E2 -26002.807} C_VEL
LIN {X 0,Y 112.459,Z 538.233,A -85,B 0,C 180,E1 -26009.153,E2 -26009.153} C_VEL
LIN {X 0,Y 112.339,Z 538.086,A -85,B 0,C 180,E1 -26013.586,E2 -26013.586} C_VEL
LIN {X 0,Y 112.511,Z 536.758,A -85,B 0,C 180,E1 -26020.8,E2 -26020.8} C_VEL
LIN {X 0,Y 113.968,Z 534.167,A -85,B 0,C 180,E1 -26027.958,E2 -26027.958} C_VEL
LIN {X 0,Y 116.974,Z 530.276,A -85,B 0,C 180,E1 -26034.871,E2 -26034.871} C_VEL
LIN {X 0,Y 121.492,Z 524.988,A -85,B 0,C 180,E1 -26041.374,E2 -26041.374} C_VEL
LIN {X 0,Y 127.453,Z 518.17,A -85,B 0,C 180,E1 -26047.341,E2 -26047.341} C_VEL
LIN {X 0,Y 133.623,Z 510.754,A -85,B 0,C 180,E1 -26052.113,E2 -26052.113} C_VEL
LIN {X 0,Y 140.566,Z 501.782,A -85,B 0,C 180,E1 -26056.466,E2 -26056.466} C_VEL
LIN {X 0,Y 147.266,Z 492.578,A -85,B 0,C 180,E1 -26059.78,E2 -26059.78} C_VEL
LIN {X 0,Y 154.234,Z 481.914,A -85,B 0,C 180,E1 -26062.732,E2 -26062.732} C_VEL
LIN {X 0,Y 155.312,Z 479.539,A -85,B 0,C 180,E1 -26063.475,E2 -26063.475} C_VEL
LIN {X 0,Y 157.642,Z 471.628,A -85,B 0,C 180,E1 -26066.158,E2 -26066.158} C_VEL
LIN {X 0,Y 157.21,Z 463.869,A -85,B 0,C 180,E1 -26069.957,E2 -26069.957} C_VEL
LIN {X 0,Y 156.07,Z 456.167,A -85,B 0,C 180,E1 -26074.24,E2 -26074.24} C_VEL
LIN {X 0,Y 154.623,Z 449.274,A -85,B 0,C 180,E1 -26078.678,E2 -26078.678} C_VEL
LIN {X 0,Y 153.211,Z 444.249,A -85,B 0,C 180,E1 -26082.653,E2 -26082.653} C_VEL
LIN {X 0,Y 152.005,Z 440.135,A -85,B 0,C 180,E1 -26086.634,E2 -26086.634} C_VEL
LIN {X 0,Y 150.718,Z 435.987,A -85,B 0,C 180,E1 -26091.959,E2 -26091.959} C_VEL
LIN {X 0,Y 150.459,Z 435.499,A -85,B 0,C 180,E1 -26093.045,E2 -26093.045} C_VEL
LIN {X 0,Y 149.789,Z 435.19,A -85,B 0,C 180,E1 -26095.282,E2 -26095.282} C_VEL
LIN {X 0,Y 148.896,Z 435.909,A -85,B 0,C 180,E1 -26097.524,E2 -26097.524} C_VEL
LIN {X 0,Y 146.974,Z 439.299,A -85,B 0,C 180,E1 -26103.585,E2 -26103.585} C_VEL
LIN {X 0,Y 146.919,Z 439.729,A -85,B 0,C 180,E1 -26105.148,E2 -26105.148} C_VEL
LIN {X 0,Y 147.675,Z 441.346,A -85,B 0,C 180,E1 -26110.975,E2 -26110.975} C_VEL
LIN {X 0,Y 148.782,Z 444.868,A -85,B 0,C 180,E1 -26116.465,E2 -26116.465} C_VEL
LIN {X 0,Y 149.832,Z 448.512,A -85,B 0,C 180,E1 -26120.596,E2 -26120.596} C_VEL
LIN {X 0,Y 150.869,Z 453.351,A -85,B 0,C 180,E1 -26124.788,E2 -26124.788} C_VEL
LIN {X 0,Y 151.641,Z 458.147,A -85,B 0,C 180,E1 -26128.287,E2 -26128.287} C_VEL
LIN {X 0,Y 152.115,Z 463.59,A -85,B 0,C 180,E1 -26131.746,E2 -26131.746} C_VEL
LIN {X 0,Y 152.009,Z 468.55,A -85,B 0,C 180,E1 -26134.496,E2 -26134.496} C_VEL
LIN {X 0,Y 150.659,Z 475.056,A -85,B 0,C 180,E1 -26137.531,E2 -26137.531} C_VEL
LIN {X 0,Y 149.789,Z 477.811,A -85,B 0,C 180,E1 -26138.702,E2 -26138.702} C_VEL
LIN {X 0,Y 142.089,Z 488.757,A -85,B 0,C 180,E1 -26142.104,E2 -26142.104} C_VEL
LIN {X 0,Y 135.388,Z 497.131,A -85,B 0,C 180,E1 -26145.51,E2 -26145.51} C_VEL
LIN {X 0,Y 128.126,Z 505.341,A -85,B 0,C 180,E1 -26150.011,E2 -26150.011} C_VEL
LIN {X 0,Y 122.107,Z 511.771,A -85,B 0,C 180,E1 -26154.861,E2 -26154.861} C_VEL
LIN {X 0,Y 115.847,Z 517.713,A -85,B 0,C 180,E1 -26160.966,E2 -26160.966} C_VEL
LIN {X 0,Y 111.204,Z 522.139,A -85,B 0,C 180,E1 -26167.716,E2 -26167.716} C_VEL
LIN {X 0,Y 107.926,Z 525.218,A -85,B 0,C 180,E1 -26174.902,E2 -26174.902} C_VEL
LIN {X 0,Y 106.106,Z 527.038,A -85,B 0,C 180,E1 -26182.388,E2 -26182.388} C_VEL
LIN {X 0,Y 105.55,Z 527.648,A -85,B 0,C 180,E1 -26190,E2 -26190} C_VEL
LIN {X 0,Y 106.106,Z 527.069,A -85,B 0,C 180,E1 -26197.613,E2 -26197.613} C_VEL
LIN {X 0,Y 107.896,Z 525.289,A -85,B 0,C 180,E1 -26205.103,E2 -26205.103} C_VEL
LIN {X 0,Y 111.178,Z 522.242,A -85,B 0,C 180,E1 -26212.29,E2 -26212.29} C_VEL
LIN {X 0,Y 115.788,Z 517.854,A -85,B 0,C 180,E1 -26219.051,E2 -26219.051} C_VEL
LIN {X 0,Y 122.085,Z 511.969,A -85,B 0,C 180,E1 -26225.147,E2 -26225.147} C_VEL
LIN {X 0,Y 127.953,Z 505.697,A -85,B 0,C 180,E1 -26229.933,E2 -26229.933} C_VEL
LIN {X 0,Y 135.303,Z 497.421,A -85,B 0,C 180,E1 -26234.526,E2 -26234.526} C_VEL
LIN {X 0,Y 142.019,Z 489.098,A -85,B 0,C 180,E1 -26237.928,E2 -26237.928} C_VEL
LIN {X 0,Y 147.84,Z 481.018,A -85,B 0,C 180,E1 -26240.534,E2 -26240.534} C_VEL
LIN {X 0,Y 149.815,Z 478.184,A -85,B 0,C 180,E1 -26241.313,E2 -26241.313} C_VEL
LIN {X 0,Y 150.86,Z 474.882,A -85,B 0,C 180,E1 -26242.726,E2 -26242.726} C_VEL
LIN {X 0,Y 152.065,Z 468.939,A -85,B 0,C 180,E1 -26245.518,E2 -26245.518} C_VEL
LIN {X 0,Y 152.263,Z 464.106,A -85,B 0,C 180,E1 -26248.15,E2 -26248.15} C_VEL
LIN {X 0,Y 151.663,Z 457.528,A -85,B 0,C 180,E1 -26252.393,E2 -26252.393} C_VEL
LIN {X 0,Y 150.717,Z 451.904,A -85,B 0,C 180,E1 -26256.649,E2 -26256.649} C_VEL
LIN {X 0,Y 149.609,Z 447.547,A -85,B 0,C 180,E1 -26260.802,E2 -26260.802} C_VEL
LIN {X 0,Y 148.919,Z 445.26,A -85,B 0,C 180,E1 -26263.551,E2 -26263.551} C_VEL
LIN {X 0,Y 147.857,Z 441.67,A -85,B 0,C 180,E1 -26269.039,E2 -26269.039} C_VEL
LIN {X 0,Y 147.427,Z 440.669,A -85,B 0,C 180,E1 -26271.777,E2 -26271.777} C_VEL
LIN {X 0,Y 147.064,Z 439.709,A -85,B 0,C 180,E1 -26277.26,E2 -26277.26} C_VEL
LIN {X 0,Y 147.122,Z 439.764,A -85,B 0,C 180,E1 -26280,E2 -26280} C_VEL
LIN {X 0,Y 147.413,Z 441.545,A -85,B 0,C 180,E1 -26285.471,E2 -26285.471} C_VEL
LIN {X 0,Y 147.86,Z 442.84,A -85,B 0,C 180,E1 -26288.198,E2 -26288.198} C_VEL
LIN {X 0,Y 148.916,Z 447.127,A -85,B 0,C 180,E1 -26293.648,E2 -26293.648} C_VEL
LIN {X 0,Y 149.866,Z 451.406,A -85,B 0,C 180,E1 -26297.747,E2 -26297.747} C_VEL
LIN {X 0,Y 151.03,Z 457.75,A -85,B 0,C 180,E1 -26302.575,E2 -26302.575} C_VEL
LIN {X 0,Y 151.863,Z 464.142,A -85,B 0,C 180,E1 -26306.663,E2 -26306.663} C_VEL
LIN {X 0,Y 152.317,Z 470.927,A -85,B 0,C 180,E1 -26310.5,E2 -26310.5} C_VEL
LIN {X 0,Y 152.284,Z 475.047,A -85,B 0,C 180,E1 -26312.621,E2 -26312.621} C_VEL
LIN {X 0,Y 149.59,Z 482.429,A -85,B 0,C 180,E1 -26315.245,E2 -26315.245} C_VEL
LIN {X 0,Y 142.763,Z 492.428,A -85,B 0,C 180,E1 -26318.032,E2 -26318.032} C_VEL
LIN {X 0,Y 134.656,Z 502.979,A -85,B 0,C 180,E1 -26321.948,E2 -26321.948} C_VEL
LIN {X 0,Y 127.445,Z 511.695,A -85,B 0,C 180,E1 -26326.423,E2 -26326.423} C_VEL
LIN {X 0,Y 121.858,Z 517.948,A -85,B 0,C 180,E1 -26330.623,E2 -26330.623} C_VEL
LIN {X 0,Y 115.407,Z 524.733,A -85,B 0,C 180,E1 -26336.764,E2 -26336.764} C_VEL
LIN {X 0,Y 110.577,Z 530.001,A -85,B 0,C 180,E1 -26343.582,E2 -26343.582} C_VEL
LIN {X 0,Y 107.192,Z 533.874,A -85,B 0,C 180,E1 -26350.863,E2 -26350.863} C_VEL
LIN {X 0,Y 105.486,Z 536.442,A -85,B 0,C 180,E1 -26358.47,E2 -26358.47} C_VEL
LIN {X 0,Y 105.238,Z 537.747,A -85,B 0,C 180,E1 -26366.17,E2 -26366.17} C_VEL
LIN {X 0,Y 105.419,Z 537.92,A -85,B 0,C 180,E1 -26370,E2 -26370} C_VEL
LIN {X 0,Y 105.238,Z 537.74,A -85,B 0,C 180,E1 -26373.829,E2 -26373.829} C_VEL
LIN {X 0,Y 105.496,Z 536.41,A -85,B 0,C 180,E1 -26381.528,E2 -26381.528} C_VEL
LIN {X 0,Y 107.173,Z 533.818,A -85,B 0,C 180,E1 -26389.14,E2 -26389.14} C_VEL
LIN {X 0,Y 110.479,Z 529.924,A -85,B 0,C 180,E1 -26396.442,E2 -26396.442} C_VEL
LIN {X 0,Y 115.398,Z 524.633,A -85,B 0,C 180,E1 -26403.238,E2 -26403.238} C_VEL
LIN {X 0,Y 121.835,Z 517.813,A -85,B 0,C 180,E1 -26409.385,E2 -26409.385} C_VEL
LIN {X 0,Y 128.372,Z 510.389,A -85,B 0,C 180,E1 -26414.269,E2 -26414.269} C_VEL
LIN {X 0,Y 135.725,Z 501.409,A -85,B 0,C 180,E1 -26418.662,E2 -26418.662} C_VEL
LIN {X 0,Y 142.735,Z 492.191,A -85,B 0,C 180,E1 -26421.981,E2 -26421.981} C_VEL
LIN {X 0,Y 149.537,Z 482.174,A -85,B 0,C 180,E1 -26424.766,E2 -26424.766} C_VEL
LIN {X 0,Y 151.938,Z 475.473,A -85,B 0,C 180,E1 -26427.172,E2 -26427.172} C_VEL
LIN {X 0,Y 152.251,Z 472.311,A -85,B 0,C 180,E1 -26428.657,E2 -26428.657} C_VEL
LIN {X 0,Y 151.921,Z 465.393,A -85,B 0,C 180,E1 -26432.445,E2 -26432.445} C_VEL
LIN {X 0,Y 151.06,Z 458.572,A -85,B 0,C 180,E1 -26436.706,E2 -26436.706} C_VEL
LIN {X 0,Y 150.044,Z 452.897,A -85,B 0,C 180,E1 -26440.861,E2 -26440.861} C_VEL
LIN {X 0,Y 149.336,Z 449.698,A -85,B 0,C 180,E1 -26443.599,E2 -26443.599} C_VEL
LIN {X 0,Y 148.753,Z 446.875,A -85,B 0,C 180,E1 -26446.336,E2 -26446.336} C_VEL
LIN {X 0,Y 147.64,Z 442.669,A -85,B 0,C 180,E1 -26451.79,E2 -26451.79} C_VEL
LIN {X 0,Y 146.937,Z 440.336,A -85,B 0,C 180,E1 -26457.259,E2 -26457.259} C_VEL
LIN {X 0,Y 146.956,Z 439.434,A -85,B 0,C 180,E1 -26460,E2 -26460} C_VEL
LIN {X 0,Y 146.894,Z 439.381,A -85,B 0,C 180,E1 -26462.743,E2 -26462.743} C_VEL
LIN {X 0,Y 146.919,Z 439.729,A -85,B 0,C 180,E1 -26465.148,E2 -26465.148} C_VEL
LIN {X 0,Y 146.82,Z 440.815,A -85,B 0,C 180,E1 -26467.407,E2 -26467.407} C_VEL
LIN {X 0,Y 146.368,Z 442.975,A -85,B 0,C 180,E1 -26469.567,E2 -26469.567} C_VEL
LIN {X 0,Y 145.032,Z 450.111,A -85,B 0,C 180,E1 -26475.242,E2 -26475.242} C_VEL
LIN {X 0,Y 145.182,Z 451.416,A -85,B 0,C 180,E1 -26476.749,E2 -26476.749} C_VEL
LIN {X 0,Y 145.905,Z 454.815,A -85,B 0,C 180,E1 -26480.628,E2 -26480.628} C_VEL
LIN {X 0,Y 146.506,Z 458.877,A -85,B 0,C 180,E1 -26484.294,E2 -26484.294} C_VEL
LIN {X 0,Y 146.928,Z 463.466,A -85,B 0,C 180,E1 -26487.799,E2 -26487.799} C_VEL
LIN {X 0,Y 147.012,Z 469.353,A -85,B 0,C 180,E1 -26491.727,E2 -26491.727} C_VEL
LIN {X 0,Y 146.493,Z 473.191,A -85,B 0,C 180,E1 -26493.844,E2 -26493.844} C_VEL
LIN {X 0,Y 145.087,Z 478.267,A -85,B 0,C 180,E1 -26496.338,E2 -26496.338} C_VEL
LIN {X 0,Y 144.29,Z 479.891,A -85,B 0,C 180,E1 -26497.001,E2 -26497.001} C_VEL
LIN {X 0,Y 137.435,Z 489.132,A -85,B 0,C 180,E1 -26499.91,E2 -26499.91} C_VEL
LIN {X 0,Y 130.416,Z 497.497,A -85,B 0,C 180,E1 -26503.322,E2 -26503.322} C_VEL
LIN {X 0,Y 122.618,Z 505.841,A -85,B 0,C 180,E1 -26507.977,E2 -26507.977} C_VEL
LIN {X 0,Y 116.374,Z 512.124,A -85,B 0,C 180,E1 -26512.849,E2 -26512.849} C_VEL
LIN {X 0,Y 109.685,Z 518.062,A -85,B 0,C 180,E1 -26519.163,E2 -26519.163} C_VEL
LIN {X 0,Y 104.678,Z 522.485,A -85,B 0,C 180,E1 -26526.245,E2 -26526.245} C_VEL
LIN {X 0,Y 101.089,Z 525.564,A -85,B 0,C 180,E1 -26533.854,E2 -26533.854} C_VEL
LIN {X 0,Y 99.077,Z 527.383,A -85,B 0,C 180,E1 -26541.844,E2 -26541.844} C_VEL
LIN {X 0,Y 98.482,Z 527.992,A -85,B 0,C 180,E1 -26550,E2 -26550} C_VEL
LIN {X 0,Y 99.077,Z 527.414,A -85,B 0,C 180,E1 -26558.157,E2 -26558.157} C_VEL
LIN {X 0,Y 101.046,Z 525.634,A -85,B 0,C 180,E1 -26566.154,E2 -26566.154} C_VEL
LIN {X 0,Y 104.637,Z 522.587,A -85,B 0,C 180,E1 -26573.766,E2 -26573.766} C_VEL
LIN {X 0,Y 109.633,Z 518.199,A -85,B 0,C 180,E1 -26580.854,E2 -26580.854} C_VEL
LIN {X 0,Y 116.35,Z 512.318,A -85,B 0,C 180,E1 -26587.16,E2 -26587.16} C_VEL
LIN {X 0,Y 122.847,Z 505.797,A -85,B 0,C 180,E1 -26592.238,E2 -26592.238} C_VEL
LIN {X 0,Y 130.348,Z 497.78,A -85,B 0,C 180,E1 -26596.71,E2 -26596.71} C_VEL
LIN {X 0,Y 137.354,Z 489.469,A -85,B 0,C 180,E1 -26600.131,E2 -26600.131} C_VEL
LIN {X 0,Y 144.25,Z 480.268,A -85,B 0,C 180,E1 -26603.037,E2 -26603.037} C_VEL
LIN {X 0,Y 145.136,Z 478.642,A -85,B 0,C 180,E1 -26603.655,E2 -26603.655} C_VEL
LIN {X 0,Y 146.781,Z 472.498,A -85,B 0,C 180,E1 -26606.704,E2 -26606.704} C_VEL
LIN {X 0,Y 147.19,Z 468.151,A -85,B 0,C 180,E1 -26609.257,E2 -26609.257} C_VEL
LIN {X 0,Y 146.93,Z 461.725,A -85,B 0,C 180,E1 -26613.739,E2 -26613.739} C_VEL
LIN {X 0,Y 146.439,Z 457.191,A -85,B 0,C 180,E1 -26617.421,E2 -26617.421} C_VEL
LIN {X 0,Y 145.62,Z 452.979,A -85,B 0,C 180,E1 -26621.717,E2 -26621.717} C_VEL
LIN {X 0,Y 144.801,Z 449.84,A -85,B 0,C 180,E1 -26626.102,E2 -26626.102} C_VEL
LIN {X 0,Y 144.478,Z 448.211,A -85,B 0,C 180,E1 -26628.78,E2 -26628.78} C_VEL
LIN {X 0,Y 144.163,Z 447.078,A -85,B 0,C 180,E1 -26631.59,E2 -26631.59} C_VEL
LIN {X 0,Y 143.888,Z 446.052,A -85,B 0,C 180,E1 -26637.2,E2 -26637.2} C_VEL
LIN {X 0,Y 143.932,Z 446.141,A -85,B 0,C 180,E1 -26639.999,E2 -26639.999} C_VEL
LIN {X 0,Y 144.146,Z 447.95,A -85,B 0,C 180,E1 -26645.595,E2 -26645.595} C_VEL
LIN {X 0,Y 144.464,Z 449.4,A -85,B 0,C 180,E1 -26648.392,E2 -26648.392} C_VEL
LIN {X 0,Y 145.057,Z 452.545,A -85,B 0,C 180,E1 -26652.593,E2 -26652.593} C_VEL
LIN {X 0,Y 145.728,Z 456.672,A -85,B 0,C 180,E1 -26656.819,E2 -26656.819} C_VEL
LIN {X 0,Y 146.489,Z 462.78,A -85,B 0,C 180,E1 -26661.751,E2 -26661.751} C_VEL
LIN {X 0,Y 146.964,Z 469.445,A -85,B 0,C 180,E1 -26666.253,E2 -26666.253} C_VEL
LIN {X 0,Y 146.992,Z 475.329,A -85,B 0,C 180,E1 -26669.764,E2 -26669.764} C_VEL
LIN {X 0,Y 146.661,Z 478.453,A -85,B 0,C 180,E1 -26671.392,E2 -26671.392} C_VEL
LIN {X 0,Y 144.377,Z 483.877,A -85,B 0,C 180,E1 -26673.409,E2 -26673.409} C_VEL
LIN {X 0,Y 137.217,Z 493.691,A -85,B 0,C 180,E1 -26676.225,E2 -26676.225} C_VEL
LIN {X 0,Y 129.983,Z 502.611,A -85,B 0,C 180,E1 -26679.602,E2 -26679.602} C_VEL
LIN {X 0,Y 123.819,Z 509.672,A -85,B 0,C 180,E1 -26683.097,E2 -26683.097} C_VEL
LIN {X 0,Y 116.409,Z 517.595,A -85,B 0,C 180,E1 -26688.385,E2 -26688.385} C_VEL
LIN {X 0,Y 109.467,Z 524.381,A -85,B 0,C 180,E1 -26694.702,E2 -26694.702} C_VEL
LIN {X 0,Y 104.18,Z 529.651,A -85,B 0,C 180,E1 -26701.821,E2 -26701.821} C_VEL
LIN {X 0,Y 100.455,Z 533.526,A -85,B 0,C 180,E1 -26709.524,E2 -26709.524} C_VEL
LIN {X 0,Y 98.474,Z 536.093,A -85,B 0,C 180,E1 -26717.636,E2 -26717.636} C_VEL
LIN {X 0,Y 98.122,Z 537.4,A -85,B 0,C 180,E1 -26725.892,E2 -26725.892} C_VEL
LIN {X 0,Y 98.331,Z 537.575,A -85,B 0,C 180,E1 -26730,E2 -26730} C_VEL
LIN {X 0,Y 98.123,Z 537.392,A -85,B 0,C 180,E1 -26734.107,E2 -26734.107} C_VEL
LIN {X 0,Y 98.481,Z 536.061,A -85,B 0,C 180,E1 -26742.362,E2 -26742.362} C_VEL
LIN {X 0,Y 100.433,Z 533.469,A -85,B 0,C 180,E1 -26750.48,E2 -26750.48} C_VEL
LIN {X 0,Y 104.091,Z 529.572,A -85,B 0,C 180,E1 -26758.205,E2 -26758.205} C_VEL
LIN {X 0,Y 109.46,Z 524.279,A -85,B 0,C 180,E1 -26765.3,E2 -26765.3} C_VEL
LIN {X 0,Y 116.385,Z 517.456,A -85,B 0,C 180,E1 -26771.624,E2 -26771.624} C_VEL
LIN {X 0,Y 123.551,Z 509.739,A -85,B 0,C 180,E1 -26776.787,E2 -26776.787} C_VEL
LIN {X 0,Y 131.109,Z 501.037,A -85,B 0,C 180,E1 -26781.011,E2 -26781.011} C_VEL
LIN {X 0,Y 138.419,Z 491.802,A -85,B 0,C 180,E1 -26784.329,E2 -26784.329} C_VEL
LIN {X 0,Y 144.33,Z 483.61,A -85,B 0,C 180,E1 -26786.604,E2 -26786.604} C_VEL
LIN {X 0,Y 146.533,Z 478.274,A -85,B 0,C 180,E1 -26788.603,E2 -26788.603} C_VEL
LIN {X 0,Y 146.85,Z 476.438,A -85,B 0,C 180,E1 -26789.48,E2 -26789.48} C_VEL
LIN {X 0,Y 146.92,Z 470.437,A -85,B 0,C 180,E1 -26792.972,E2 -26792.972} C_VEL
LIN {X 0,Y 146.484,Z 463.664,A -85,B 0,C 180,E1 -26797.43,E2 -26797.43} C_VEL
LIN {X 0,Y 145.798,Z 458.114,A -85,B 0,C 180,E1 -26801.741,E2 -26801.741} C_VEL
LIN {X 0,Y 145.283,Z 454.897,A -85,B 0,C 180,E1 -26804.714,E2 -26804.714} C_VEL
LIN {X 0,Y 144.609,Z 451.254,A -85,B 0,C 180,E1 -26808.791,E2 -26808.791} C_VEL
LIN {X 0,Y 144.27,Z 449.202,A -85,B 0,C 180,E1 -26811.597,E2 -26811.597} C_VEL
LIN {X 0,Y 143.933,Z 447.768,A -85,B 0,C 180,E1 -26814.396,E2 -26814.396} C_VEL
LIN {X 0,Y 143.778,Z 445.814,A -85,B 0,C 180,E1 -26820.001,E2 -26820.001} C_VEL
LIN {X 0,Y 143.727,Z 445.732,A -85,B 0,C 180,E1 -26822.803,E2 -26822.803} C_VEL
LIN {X 0,Y 143.971,Z 446.812,A -85,B 0,C 180,E1 -26828.422,E2 -26828.422} C_VEL
LIN {X 0,Y 144.326,Z 447.868,A -85,B 0,C 180,E1 -26831.232,E2 -26831.232} C_VEL
LIN {X 0,Y 144.703,Z 449.525,A -85,B 0,C 180,E1 -26834.055,E2 -26834.055} C_VEL
LIN {X 0,Y 145.182,Z 451.416,A -85,B 0,C 180,E1 -26836.749,E2 -26836.749} C_VEL
LIN {X 0,Y 145.331,Z 452.789,A -85,B 0,C 180,E1 -26838.197,E2 -26838.197} C_VEL
LIN {X 0,Y 145.143,Z 454.663,A -85,B 0,C 180,E1 -26839.56,E2 -26839.56} C_VEL
LIN {X 0,Y 144.446,Z 458.057,A -85,B 0,C 180,E1 -26841.483,E2 -26841.483} C_VEL
LIN {X 0,Y 142.269,Z 466.624,A -85,B 0,C 180,E1 -26845.941,E2 -26845.941} C_VEL
LIN {X 0,Y 142.037,Z 468.693,A -85,B 0,C 180,E1 -26847.348,E2 -26847.348} C_VEL
LIN {X 0,Y 141.808,Z 473.415,A -85,B 0,C 180,E1 -26850.7,E2 -26850.7} C_VEL
LIN {X 0,Y 140.725,Z 477.972,A -85,B 0,C 180,E1 -26853.323,E2 -26853.323} C_VEL
LIN {X 0,Y 139.623,Z 480.868,A -85,B 0,C 180,E1 -26854.793,E2 -26854.793} C_VEL
LIN {X 0,Y 131.752,Z 490.977,A -85,B 0,C 180,E1 -26858.112,E2 -26858.112} C_VEL
LIN {X 0,Y 123.304,Z 500.295,A -85,B 0,C 180,E1 -26862.186,E2 -26862.186} C_VEL
LIN {X 0,Y 115.727,Z 507.8,A -85,B 0,C 180,E1 -26866.783,E2 -26866.783} C_VEL
LIN {X 0,Y 108.892,Z 514.073,A -85,B 0,C 180,E1 -26872.183,E2 -26872.183} C_VEL
LIN {X 0,Y 102.147,Z 519.621,A -85,B 0,C 180,E1 -26878.935,E2 -26878.935} C_VEL
LIN {X 0,Y 98.217,Z 522.831,A -85,B 0,C 180,E1 -26884.575,E2 -26884.575} C_VEL
LIN {X 0,Y 94.284,Z 525.91,A -85,B 0,C 180,E1 -26892.653,E2 -26892.653} C_VEL
LIN {X 0,Y 92.069,Z 527.728,A -85,B 0,C 180,E1 -26901.219,E2 -26901.219} C_VEL
LIN {X 0,Y 91.405,Z 528.337,A -85,B 0,C 180,E1 -26910,E2 -26910} C_VEL
LIN {X 0,Y 92.069,Z 527.759,A -85,B 0,C 180,E1 -26918.782,E2 -26918.782} C_VEL
LIN {X 0,Y 94.248,Z 525.979,A -85,B 0,C 180,E1 -26927.355,E2 -26927.355} C_VEL
LIN {X 0,Y 98.16,Z 522.933,A -85,B 0,C 180,E1 -26935.442,E2 -26935.442} C_VEL
LIN {X 0,Y 103.605,Z 518.545,A -85,B 0,C 180,E1 -26942.867,E2 -26942.867} C_VEL
LIN {X 0,Y 110.769,Z 512.667,A -85,B 0,C 180,E1 -26949.382,E2 -26949.382} C_VEL
LIN {X 0,Y 117.575,Z 506.248,A -85,B 0,C 180,E1 -26954.497,E2 -26954.497} C_VEL
LIN {X 0,Y 125.599,Z 498.139,A -85,B 0,C 180,E1 -26959.062,E2 -26959.062} C_VEL
LIN {X 0,Y 132.91,Z 489.84,A -85,B 0,C 180,E1 -26962.484,E2 -26962.484} C_VEL
LIN {X 0,Y 139.63,Z 481.245,A -85,B 0,C 180,E1 -26965.213,E2 -26965.213} C_VEL
LIN {X 0,Y 141.321,Z 476.4,A -85,B 0,C 180,E1 -26967.719,E2 -26967.719} C_VEL
LIN {X 0,Y 142.026,Z 472.197,A -85,B 0,C 180,E1 -26970.34,E2 -26970.34} C_VEL
LIN {X 0,Y 142.147,Z 466.33,A -85,B 0,C 180,E1 -26974.734,E2 -26974.734} C_VEL
LIN {X 0,Y 142.006,Z 462.342,A -85,B 0,C 180,E1 -26978.211,E2 -26978.211} C_VEL
LIN {X 0,Y 141.467,Z 458.324,A -85,B 0,C 180,E1 -26982.657,E2 -26982.657} C_VEL
LIN {X 0,Y 140.809,Z 454.593,A -85,B 0,C 180,E1 -26988.483,E2 -26988.483} C_VEL
LIN {X 0,Y 140.612,Z 453.348,A -85,B 0,C 180,E1 -26991.376,E2 -26991.376} C_VEL
LIN {X 0,Y 140.422,Z 452.269,A -85,B 0,C 180,E1 -26997.131,E2 -26997.131} C_VEL
LIN {X 0,Y 140.456,Z 452.378,A -85,B 0,C 180,E1 -26999.999,E2 -26999.999} C_VEL
LIN {X 0,Y 140.57,Z 454.252,A -85,B 0,C 180,E1 -27005.738,E2 -27005.738} C_VEL
LIN {X 0,Y 140.851,Z 456.843,A -85,B 0,C 180,E1 -27010.057,E2 -27010.057} C_VEL
LIN {X 0,Y 141.294,Z 460.431,A -85,B 0,C 180,E1 -27014.4,E2 -27014.4} C_VEL
LIN {X 0,Y 141.559,Z 463.391,A -85,B 0,C 180,E1 -27017.33,E2 -27017.33} C_VEL
LIN {X 0,Y 141.855,Z 468.854,A -85,B 0,C 180,E1 -27021.812,E2 -27021.812} C_VEL
LIN {X 0,Y 141.892,Z 474.086,A -85,B 0,C 180,E1 -27025.507,E2 -27025.507} C_VEL
LIN {X 0,Y 141.572,Z 479.529,A -85,B 0,C 180,E1 -27028.947,E2 -27028.947} C_VEL
LIN {X 0,Y 141.295,Z 481.08,A -85,B 0,C 180,E1 -27029.828,E2 -27029.828} C_VEL
LIN {X 0,Y 139.699,Z 484.627,A -85,B 0,C 180,E1 -27031.212,E2 -27031.212} C_VEL
LIN {X 0,Y 131.807,Z 494.947,A -85,B 0,C 180,E1 -27034.261,E2 -27034.261} C_VEL
LIN {X 0,Y 123.094,Z 504.935,A -85,B 0,C 180,E1 -27038.273,E2 -27038.273} C_VEL
LIN {X 0,Y 115.259,Z 513.202,A -85,B 0,C 180,E1 -27042.969,E2 -27042.969} C_VEL
LIN {X 0,Y 109.125,Z 519.084,A -85,B 0,C 180,E1 -27047.449,E2 -27047.449} C_VEL
LIN {X 0,Y 102.084,Z 525.492,A -85,B 0,C 180,E1 -27054.183,E2 -27054.183} C_VEL
LIN {X 0,Y 96.728,Z 530.406,A -85,B 0,C 180,E1 -27061.817,E2 -27061.817} C_VEL
LIN {X 0,Y 93.756,Z 533.177,A -85,B 0,C 180,E1 -27067.987,E2 -27067.987} C_VEL
LIN {X 0,Y 91.498,Z 535.745,A -85,B 0,C 180,E1 -27076.677,E2 -27076.677} C_VEL
LIN {X 0,Y 91.013,Z 537.053,A -85,B 0,C 180,E1 -27085.571,E2 -27085.571} C_VEL
LIN {X 0,Y 91.244,Z 537.23,A -85,B 0,C 180,E1 -27090,E2 -27090} C_VEL
LIN {X 0,Y 91.014,Z 537.045,A -85,B 0,C 180,E1 -27094.428,E2 -27094.428} C_VEL
LIN {X 0,Y 91.503,Z 535.713,A -85,B 0,C 180,E1 -27103.321,E2 -27103.321} C_VEL
LIN {X 0,Y 93.731,Z 533.118,A -85,B 0,C 180,E1 -27112.018,E2 -27112.018} C_VEL
LIN {X 0,Y 98.232,Z 528.852,A -85,B 0,C 180,E1 -27120.848,E2 -27120.848} C_VEL
LIN {X 0,Y 103.673,Z 523.926,A -85,B 0,C 180,E1 -27127.597,E2 -27127.597} C_VEL
LIN {X 0,Y 111.108,Z 517.098,A -85,B 0,C 180,E1 -27134.09,E2 -27134.09} C_VEL
LIN {X 0,Y 119.04,Z 509.066,A -85,B 0,C 180,E1 -27139.502,E2 -27139.502} C_VEL
LIN {X 0,Y 126.718,Z 500.664,A -85,B 0,C 180,E1 -27143.533,E2 -27143.533} C_VEL
LIN {X 0,Y 134.353,Z 491.415,A -85,B 0,C 180,E1 -27146.82,E2 -27146.82} C_VEL
LIN {X 0,Y 139.668,Z 484.341,A -85,B 0,C 180,E1 -27148.808,E2 -27148.808} C_VEL
LIN {X 0,Y 141.162,Z 480.957,A -85,B 0,C 180,E1 -27150.141,E2 -27150.141} C_VEL
LIN {X 0,Y 141.702,Z 476.599,A -85,B 0,C 180,E1 -27152.694,E2 -27152.694} C_VEL
LIN {X 0,Y 141.798,Z 470.732,A -85,B 0,C 180,E1 -27156.641,E2 -27156.641} C_VEL
LIN {X 0,Y 141.523,Z 464.371,A -85,B 0,C 180,E1 -27161.6,E2 -27161.6} C_VEL
LIN {X 0,Y 141.138,Z 460.237,A -85,B 0,C 180,E1 -27165.584,E2 -27165.584} C_VEL
LIN {X 0,Y 140.689,Z 456.622,A -85,B 0,C 180,E1 -27169.931,E2 -27169.931} C_VEL
LIN {X 0,Y 140.604,Z 455.592,A -85,B 0,C 180,E1 -27171.376,E2 -27171.376} C_VEL
LIN {X 0,Y 140.373,Z 454.067,A -85,B 0,C 180,E1 -27174.254,E2 -27174.254} C_VEL
LIN {X 0,Y 140.317,Z 452.057,A -85,B 0,C 180,E1 -27180.001,E2 -27180.001} C_VEL
LIN {X 0,Y 140.282,Z 451.947,A -85,B 0,C 180,E1 -27182.872,E2 -27182.872} C_VEL
LIN {X 0,Y 140.433,Z 453.092,A -85,B 0,C 180,E1 -27188.635,E2 -27188.635} C_VEL
LIN {X 0,Y 140.698,Z 454.221,A -85,B 0,C 180,E1 -27191.526,E2 -27191.526} C_VEL
LIN {X 0,Y 141.337,Z 458.005,A -85,B 0,C 180,E1 -27197.359,E2 -27197.359} C_VEL
LIN {X 0,Y 141.667,Z 460.58,A -85,B 0,C 180,E1 -27200.321,E2 -27200.321} C_VEL
LIN {X 0,Y 142.045,Z 465.767,A -85,B 0,C 180,E1 -27205.108,E2 -27205.108} C_VEL
LIN {X 0,Y 142.037,Z 468.693,A -85,B 0,C 180,E1 -27207.348,E2 -27207.348} C_VEL
LIN {X 0,Y 141.492,Z 470.96,A -85,B 0,C 180,E1 -27208.635,E2 -27208.635} C_VEL
LIN {X 0,Y 139.7,Z 474.651,A -85,B 0,C 180,E1 -27210.017,E2 -27210.017} C_VEL
LIN {X 0,Y 134.169,Z 483.282,A -85,B 0,C 180,E1 -27212.902,E2 -27212.902} C_VEL
LIN {X 0,Y 126.205,Z 492.823,A -85,B 0,C 180,E1 -27216.151,E2 -27216.151} C_VEL
LIN {X 0,Y 117.474,Z 501.873,A -85,B 0,C 180,E1 -27220.29,E2 -27220.29} C_VEL
LIN {X 0,Y 109.456,Z 509.251,A -85,B 0,C 180,E1 -27225.066,E2 -27225.066} C_VEL
LIN {X 0,Y 103.381,Z 514.423,A -85,B 0,C 180,E1 -27229.773,E2 -27229.773} C_VEL
LIN {X 0,Y 96.123,Z 519.97,A -85,B 0,C 180,E1 -27236.746,E2 -27236.746} C_VEL
LIN {X 0,Y 91.836,Z 523.178,A -85,B 0,C 180,E1 -27242.667,E2 -27242.667} C_VEL
LIN {X 0,Y 87.537,Z 526.255,A -85,B 0,C 180,E1 -27251.268,E2 -27251.268} C_VEL
LIN {X 0,Y 85.078,Z 528.073,A -85,B 0,C 180,E1 -27260.491,E2 -27260.491} C_VEL
LIN {X 0,Y 84.337,Z 528.681,A -85,B 0,C 180,E1 -27270,E2 -27270} C_VEL
LIN {X 0,Y 85.078,Z 528.103,A -85,B 0,C 180,E1 -27279.51,E2 -27279.51} C_VEL
LIN {X 0,Y 87.507,Z 526.323,A -85,B 0,C 180,E1 -27288.74,E2 -27288.74} C_VEL
LIN {X 0,Y 91.78,Z 523.279,A -85,B 0,C 180,E1 -27297.352,E2 -27297.352} C_VEL
LIN {X 0,Y 97.723,Z 518.891,A -85,B 0,C 180,E1 -27305.124,E2 -27305.124} C_VEL
LIN {X 0,Y 105.356,Z 513.017,A -85,B 0,C 180,E1 -27311.842,E2 -27311.842} C_VEL
LIN {X 0,Y 112.733,Z 506.502,A -85,B 0,C 180,E1 -27317.098,E2 -27317.098} C_VEL
LIN {X 0,Y 121.071,Z 498.498,A -85,B 0,C 180,E1 -27321.597,E2 -27321.597} C_VEL
LIN {X 0,Y 128.716,Z 490.209,A -85,B 0,C 180,E1 -27324.987,E2 -27324.987} C_VEL
LIN {X 0,Y 133.991,Z 483.867,A -85,B 0,C 180,E1 -27327.059,E2 -27327.059} C_VEL
LIN {X 0,Y 135.103,Z 482.044,A -85,B 0,C 180,E1 -27327.779,E2 -27327.779} C_VEL
LIN {X 0,Y 136.412,Z 478.378,A -85,B 0,C 180,E1 -27329.932,E2 -27329.932} C_VEL
LIN {X 0,Y 137.097,Z 473.775,A -85,B 0,C 180,E1 -27333.349,E2 -27333.349} C_VEL
LIN {X 0,Y 137.355,Z 469.4,A -85,B 0,C 180,E1 -27337.075,E2 -27337.075} C_VEL
LIN {X 0,Y 137.285,Z 465.868,A -85,B 0,C 180,E1 -27340.704,E2 -27340.704} C_VEL
LIN {X 0,Y 137.045,Z 462.542,A -85,B 0,C 180,E1 -27345.142,E2 -27345.142} C_VEL
LIN {X 0,Y 136.855,Z 460.807,A -85,B 0,C 180,E1 -27348.146,E2 -27348.146} C_VEL
LIN {X 0,Y 136.759,Z 459.498,A -85,B 0,C 180,E1 -27351.131,E2 -27351.131} C_VEL
LIN {X 0,Y 136.662,Z 458.737,A -85,B 0,C 180,E1 -27354.096,E2 -27354.096} C_VEL
LIN {X 0,Y 136.692,Z 458.318,A -85,B 0,C 180,E1 -27357.052,E2 -27357.052} C_VEL
LIN {X 0,Y 136.711,Z 458.453,A -85,B 0,C 180,E1 -27359.999,E2 -27359.999} C_VEL
LIN {X 0,Y 136.692,Z 460.429,A -85,B 0,C 180,E1 -27365.902,E2 -27365.902} C_VEL
LIN {X 0,Y 136.837,Z 463.075,A -85,B 0,C 180,E1 -27370.355,E2 -27370.355} C_VEL
LIN {X 0,Y 137.014,Z 466.835,A -85,B 0,C 180,E1 -27374.86,E2 -27374.86} C_VEL
LIN {X 0,Y 137.027,Z 471.666,A -85,B 0,C 180,E1 -27379.372,E2 -27379.372} C_VEL
LIN {X 0,Y 136.835,Z 476.659,A -85,B 0,C 180,E1 -27383.356,E2 -27383.356} C_VEL
LIN {X 0,Y 136.137,Z 482.939,A -85,B 0,C 180,E1 -27387.685,E2 -27387.685} C_VEL
LIN {X 0,Y 135.248,Z 485.182,A -85,B 0,C 180,E1 -27388.776,E2 -27388.776} C_VEL
LIN {X 0,Y 133.373,Z 487.845,A -85,B 0,C 180,E1 -27389.603,E2 -27389.603} C_VEL
LIN {X 0,Y 125.243,Z 497.588,A -85,B 0,C 180,E1 -27392.676,E2 -27392.676} C_VEL
LIN {X 0,Y 116.314,Z 507.071,A -85,B 0,C 180,E1 -27396.811,E2 -27396.811} C_VEL
LIN {X 0,Y 108.267,Z 514.901,A -85,B 0,C 180,E1 -27401.71,E2 -27401.71} C_VEL
LIN {X 0,Y 99.94,Z 522.13,A -85,B 0,C 180,E1 -27408.082,E2 -27408.082} C_VEL
LIN {X 0,Y 93.04,Z 527.904,A -85,B 0,C 180,E1 -27415.753,E2 -27415.753} C_VEL
LIN {X 0,Y 89.226,Z 531.059,A -85,B 0,C 180,E1 -27421.796,E2 -27421.796} C_VEL
LIN {X 0,Y 85.552,Z 534.271,A -85,B 0,C 180,E1 -27430.816,E2 -27430.816} C_VEL
LIN {X 0,Y 84.005,Z 536.209,A -85,B 0,C 180,E1 -27440.367,E2 -27440.367} C_VEL
LIN {X 0,Y 83.907,Z 536.707,A -85,B 0,C 180,E1 -27445.195,E2 -27445.195} C_VEL
LIN {X 0,Y 84.142,Z 536.884,A -85,B 0,C 180,E1 -27450,E2 -27450} C_VEL
LIN {X 0,Y 83.908,Z 536.698,A -85,B 0,C 180,E1 -27454.804,E2 -27454.804} C_VEL
LIN {X 0,Y 84.546,Z 535.364,A -85,B 0,C 180,E1 -27464.44,E2 -27464.44} C_VEL
LIN {X 0,Y 87.115,Z 532.769,A -85,B 0,C 180,E1 -27473.789,E2 -27473.789} C_VEL
LIN {X 0,Y 91.719,Z 528.818,A -85,B 0,C 180,E1 -27482.556,E2 -27482.556} C_VEL
LIN {X 0,Y 98.084,Z 523.573,A -85,B 0,C 180,E1 -27490.156,E2 -27490.156} C_VEL
LIN {X 0,Y 106.06,Z 516.74,A -85,B 0,C 180,E1 -27496.795,E2 -27496.795} C_VEL
LIN {X 0,Y 113.871,Z 509.299,A -85,B 0,C 180,E1 -27501.89,E2 -27501.89} C_VEL
LIN {X 0,Y 122.597,Z 500.292,A -85,B 0,C 180,E1 -27506.225,E2 -27506.225} C_VEL
LIN {X 0,Y 130.564,Z 491.028,A -85,B 0,C 180,E1 -27509.457,E2 -27509.457} C_VEL
LIN {X 0,Y 134.316,Z 486.304,A -85,B 0,C 180,E1 -27510.755,E2 -27510.755} C_VEL
LIN {X 0,Y 135.733,Z 483.894,A -85,B 0,C 180,E1 -27511.67,E2 -27511.67} C_VEL
LIN {X 0,Y 136.241,Z 481.404,A -85,B 0,C 180,E1 -27513.168,E2 -27513.168} C_VEL
LIN {X 0,Y 136.711,Z 476.425,A -85,B 0,C 180,E1 -27516.671,E2 -27516.671} C_VEL
LIN {X 0,Y 136.901,Z 471.281,A -85,B 0,C 180,E1 -27520.767,E2 -27520.767} C_VEL
LIN {X 0,Y 136.887,Z 466.623,A -85,B 0,C 180,E1 -27525.126,E2 -27525.126} C_VEL
LIN {X 0,Y 136.686,Z 462.865,A -85,B 0,C 180,E1 -27529.633,E2 -27529.633} C_VEL
LIN {X 0,Y 136.522,Z 460.228,A -85,B 0,C 180,E1 -27534.091,E2 -27534.091} C_VEL
LIN {X 0,Y 136.582,Z 458.149,A -85,B 0,C 180,E1 -27540.001,E2 -27540.001} C_VEL
LIN {X 0,Y 136.562,Z 458.011,A -85,B 0,C 180,E1 -27542.95,E2 -27542.95} C_VEL
LIN {X 0,Y 136.611,Z 459.226,A -85,B 0,C 180,E1 -27548.879,E2 -27548.879} C_VEL
LIN {X 0,Y 136.773,Z 460.81,A -85,B 0,C 180,E1 -27552.497,E2 -27552.497} C_VEL
LIN {X 0,Y 137.066,Z 463.215,A -85,B 0,C 180,E1 -27556.381,E2 -27556.381} C_VEL
LIN {X 0,Y 137.234,Z 467.119,A -85,B 0,C 180,E1 -27561.008,E2 -27561.008} C_VEL
LIN {X 0,Y 137.215,Z 470.434,A -85,B 0,C 180,E1 -27564.19,E2 -27564.19} C_VEL
LIN {X 0,Y 136.876,Z 474.554,A -85,B 0,C 180,E1 -27567.524,E2 -27567.524} C_VEL
LIN {X 0,Y 136.363,Z 477.971,A -85,B 0,C 180,E1 -27570.037,E2 -27570.037} C_VEL
LIN {X 0,Y 135.063,Z 481.733,A -85,B 0,C 180,E1 -27572.256,E2 -27572.256} C_VEL
LIN {X 0,Y 134.169,Z 483.282,A -85,B 0,C 180,E1 -27572.902,E2 -27572.902} C_VEL
LIN {X 0,Y 132.318,Z 485.914,A -85,B 0,C 180,E1 -27573.831,E2 -27573.831} C_VEL
LIN {X 0,Y 129.903,Z 488.56,A -85,B 0,C 180,E1 -27574.505,E2 -27574.505} C_VEL
LIN {X 0,Y 124.114,Z 493.644,A -85,B 0,C 180,E1 -27575.394,E2 -27575.394} C_VEL
LIN {X 0,Y 116.267,Z 499.647,A -85,B 0,C 180,E1 -27576.578,E2 -27576.578} C_VEL
LIN {X 0,Y 112.129,Z 503.022,A -85,B 0,C 180,E1 -27577.986,E2 -27577.986} C_VEL
LIN {X 0,Y 104.539,Z 509.609,A -85,B 0,C 180,E1 -27582.31,E2 -27582.31} C_VEL
LIN {X 0,Y 98.071,Z 514.774,A -85,B 0,C 180,E1 -27587.095,E2 -27587.095} C_VEL
LIN {X 0,Y 90.266,Z 520.318,A -85,B 0,C 180,E1 -27594.272,E2 -27594.272} C_VEL
LIN {X 0,Y 85.576,Z 523.525,A -85,B 0,C 180,E1 -27600.478,E2 -27600.478} C_VEL
LIN {X 0,Y 80.859,Z 526.6,A -85,B 0,C 180,E1 -27609.656,E2 -27609.656} C_VEL
LIN {X 0,Y 78.101,Z 528.418,A -85,B 0,C 180,E1 -27619.632,E2 -27619.632} C_VEL
LIN {X 0,Y 77.272,Z 529.025,A -85,B 0,C 180,E1 -27630.001,E2 -27630.001} C_VEL
LIN {X 0,Y 78.101,Z 528.447,A -85,B 0,C 180,E1 -27640.369,E2 -27640.369} C_VEL
LIN {X 0,Y 80.807,Z 526.668,A -85,B 0,C 180,E1 -27650.359,E2 -27650.359} C_VEL
LIN {X 0,Y 85.527,Z 523.625,A -85,B 0,C 180,E1 -27659.541,E2 -27659.541} C_VEL
LIN {X 0,Y 92.016,Z 519.235,A -85,B 0,C 180,E1 -27667.664,E2 -27667.664} C_VEL
LIN {X 0,Y 100.159,Z 513.367,A -85,B 0,C 180,E1 -27674.564,E2 -27674.564} C_VEL
LIN {X 0,Y 107.901,Z 506.953,A -85,B 0,C 180,E1 -27679.792,E2 -27679.792} C_VEL
LIN {X 0,Y 116.799,Z 498.857,A -85,B 0,C 180,E1 -27684.324,E2 -27684.324} C_VEL
LIN {X 0,Y 126.153,Z 489.093,A -85,B 0,C 180,E1 -27688.167,E2 -27688.167} C_VEL
LIN {X 0,Y 130.115,Z 484.266,A -85,B 0,C 180,E1 -27689.795,E2 -27689.795} C_VEL
LIN {X 0,Y 131.412,Z 480.751,A -85,B 0,C 180,E1 -27692.098,E2 -27692.098} C_VEL
LIN {X 0,Y 132.233,Z 476.016,A -85,B 0,C 180,E1 -27696.133,E2 -27696.133} C_VEL
LIN {X 0,Y 132.633,Z 472.269,A -85,B 0,C 180,E1 -27699.853,E2 -27699.853} C_VEL
LIN {X 0,Y 132.699,Z 468.63,A -85,B 0,C 180,E1 -27704.644,E2 -27704.644} C_VEL
LIN {X 0,Y 132.607,Z 466.866,A -85,B 0,C 180,E1 -27707.76,E2 -27707.76} C_VEL
LIN {X 0,Y 132.619,Z 465.495,A -85,B 0,C 180,E1 -27710.852,E2 -27710.852} C_VEL
LIN {X 0,Y 132.626,Z 464.648,A -85,B 0,C 180,E1 -27713.916,E2 -27713.916} C_VEL
LIN {X 0,Y 132.688,Z 464.214,A -85,B 0,C 180,E1 -27716.963,E2 -27716.963} C_VEL
LIN {X 0,Y 132.705,Z 464.352,A -85,B 0,C 180,E1 -27719.999,E2 -27719.999} C_VEL
LIN {X 0,Y 132.574,Z 465.222,A -85,B 0,C 180,E1 -27723.038,E2 -27723.038} C_VEL
LIN {X 0,Y 132.534,Z 466.441,A -85,B 0,C 180,E1 -27726.087,E2 -27726.087} C_VEL
LIN {X 0,Y 132.491,Z 469.202,A -85,B 0,C 180,E1 -27730.699,E2 -27730.699} C_VEL
LIN {X 0,Y 132.355,Z 473.15,A -85,B 0,C 180,E1 -27735.396,E2 -27735.396} C_VEL
LIN {X 0,Y 131.912,Z 478.406,A -85,B 0,C 180,E1 -27740.261,E2 -27740.261} C_VEL
LIN {X 0,Y 131.219,Z 483.626,A -85,B 0,C 180,E1 -27744.422,E2 -27744.422} C_VEL
LIN {X 0,Y 130.665,Z 486.266,A -85,B 0,C 180,E1 -27746.342,E2 -27746.342} C_VEL
LIN {X 0,Y 130.215,Z 487.133,A -85,B 0,C 180,E1 -27746.753,E2 -27746.753} C_VEL
LIN {X 0,Y 121.514,Z 497.212,A -85,B 0,C 180,E1 -27749.822,E2 -27749.822} C_VEL
LIN {X 0,Y 112.148,Z 506.706,A -85,B 0,C 180,E1 -27753.865,E2 -27753.865} C_VEL
LIN {X 0,Y 103.603,Z 514.542,A -85,B 0,C 180,E1 -27758.728,E2 -27758.728} C_VEL
LIN {X 0,Y 94.72,Z 521.778,A -85,B 0,C 180,E1 -27765.179,E2 -27765.179} C_VEL
LIN {X 0,Y 87.345,Z 527.425,A -85,B 0,C 180,E1 -27772.88,E2 -27772.88} C_VEL
LIN {X 0,Y 82.975,Z 530.71,A -85,B 0,C 180,E1 -27779.455,E2 -27779.455} C_VEL
LIN {X 0,Y 78.808,Z 533.922,A -85,B 0,C 180,E1 -27789.101,E2 -27789.101} C_VEL
LIN {X 0,Y 76.958,Z 535.861,A -85,B 0,C 180,E1 -27799.475,E2 -27799.475} C_VEL
LIN {X 0,Y 77.051,Z 536.539,A -85,B 0,C 180,E1 -27809.999,E2 -27809.999} C_VEL
LIN {X 0,Y 76.961,Z 535.84,A -85,B 0,C 180,E1 -27820.523,E2 -27820.523} C_VEL
LIN {X 0,Y 78.796,Z 533.874,A -85,B 0,C 180,E1 -27830.902,E2 -27830.902} C_VEL
LIN {X 0,Y 82.908,Z 530.637,A -85,B 0,C 180,E1 -27840.571,E2 -27840.571} C_VEL
LIN {X 0,Y 88.989,Z 526.051,A -85,B 0,C 180,E1 -27849.183,E2 -27849.183} C_VEL
LIN {X 0,Y 96.794,Z 520.001,A -85,B 0,C 180,E1 -27856.558,E2 -27856.558} C_VEL
LIN {X 0,Y 104.736,Z 513.349,A -85,B 0,C 180,E1 -27862.041,E2 -27862.041} C_VEL
LIN {X 0,Y 113.422,Z 505.261,A -85,B 0,C 180,E1 -27866.773,E2 -27866.773} C_VEL
LIN {X 0,Y 122.893,Z 495.478,A -85,B 0,C 180,E1 -27870.705,E2 -27870.705} C_VEL
LIN {X 0,Y 130.142,Z 486.922,A -85,B 0,C 180,E1 -27873.242,E2 -27873.242} C_VEL
LIN {X 0,Y 130.597,Z 486.06,A -85,B 0,C 180,E1 -27873.643,E2 -27873.643} C_VEL
LIN {X 0,Y 131.369,Z 481.93,A -85,B 0,C 180,E1 -27876.657,E2 -27876.657} C_VEL
LIN {X 0,Y 131.854,Z 478.157,A -85,B 0,C 180,E1 -27879.73,E2 -27879.73} C_VEL
LIN {X 0,Y 132.233,Z 472.952,A -85,B 0,C 180,E1 -27884.59,E2 -27884.59} C_VEL
LIN {X 0,Y 132.354,Z 468.992,A -85,B 0,C 180,E1 -27889.29,E2 -27889.29} C_VEL
LIN {X 0,Y 132.379,Z 466.242,A -85,B 0,C 180,E1 -27893.905,E2 -27893.905} C_VEL
LIN {X 0,Y 132.422,Z 465.003,A -85,B 0,C 180,E1 -27896.958,E2 -27896.958} C_VEL
LIN {X 0,Y 132.578,Z 464.074,A -85,B 0,C 180,E1 -27900.001,E2 -27900.001} C_VEL
LIN {X 0,Y 132.573,Z 463.914,A -85,B 0,C 180,E1 -27903.039,E2 -27903.039} C_VEL
LIN {X 0,Y 132.449,Z 464.818,A -85,B 0,C 180,E1 -27907.692,E2 -27907.692} C_VEL
LIN {X 0,Y 132.529,Z 466.522,A -85,B 0,C 180,E1 -27912.247,E2 -27912.247} C_VEL
LIN {X 0,Y 132.617,Z 468.283,A -85,B 0,C 180,E1 -27915.366,E2 -27915.366} C_VEL
LIN {X 0,Y 132.509,Z 472,A -85,B 0,C 180,E1 -27920.167,E2 -27920.167} C_VEL
LIN {X 0,Y 131.948,Z 477.082,A -85,B 0,C 180,E1 -27925.112,E2 -27925.112} C_VEL
LIN {X 0,Y 130.951,Z 481.773,A -85,B 0,C 180,E1 -27928.884,E2 -27928.884} C_VEL
LIN {X 0,Y 130.095,Z 483.896,A -85,B 0,C 180,E1 -27930.191,E2 -27930.191} C_VEL
LIN {X 0,Y 128.952,Z 485.519,A -85,B 0,C 180,E1 -27930.864,E2 -27930.864} C_VEL
LIN {X 0,Y 120.853,Z 494.595,A -85,B 0,C 180,E1 -27934.036,E2 -27934.036} C_VEL
LIN {X 0,Y 112.129,Z 503.022,A -85,B 0,C 180,E1 -27937.986,E2 -27937.986} C_VEL
LIN {X 0,Y 108.196,Z 506.207,A -85,B 0,C 180,E1 -27939.609,E2 -27939.609} C_VEL
LIN {X 0,Y 100.624,Z 511.035,A -85,B 0,C 180,E1 -27941.905,E2 -27941.905} C_VEL
LIN {X 0,Y 93.046,Z 515.387,A -85,B 0,C 180,E1 -27944.681,E2 -27944.681} C_VEL
LIN {X 0,Y 89.23,Z 517.694,A -85,B 0,C 180,E1 -27947.114,E2 -27947.114} C_VEL
LIN {X 0,Y 82.762,Z 521.839,A -85,B 0,C 180,E1 -27953.529,E2 -27953.529} C_VEL
LIN {X 0,Y 76.61,Z 525.57,A -85,B 0,C 180,E1 -27962.698,E2 -27962.698} C_VEL
LIN {X 0,Y 72.411,Z 528.008,A -85,B 0,C 180,E1 -27973.072,E2 -27973.072} C_VEL
LIN {X 0,Y 70.382,Z 529.217,A -85,B 0,C 180,E1 -27984.27,E2 -27984.27} C_VEL
LIN {X 0,Y 70.197,Z 529.37,A -85,B 0,C 180,E1 -27990.001,E2 -27990.001} C_VEL
LIN {X 0,Y 71.132,Z 528.792,A -85,B 0,C 180,E1 -28001.398,E2 -28001.398} C_VEL
LIN {X 0,Y 74.195,Z 527.013,A -85,B 0,C 180,E1 -28012.266,E2 -28012.266} C_VEL
LIN {X 0,Y 79.424,Z 523.969,A -85,B 0,C 180,E1 -28022.069,E2 -28022.069} C_VEL
LIN {X 0,Y 86.516,Z 519.58,A -85,B 0,C 180,E1 -28030.533,E2 -28030.533} C_VEL
LIN {X 0,Y 95.211,Z 513.716,A -85,B 0,C 180,E1 -28037.575,E2 -28037.575} C_VEL
LIN {X 0,Y 103.581,Z 507.207,A -85,B 0,C 180,E1 -28042.869,E2 -28042.869} C_VEL
LIN {X 0,Y 112.819,Z 499.215,A -85,B 0,C 180,E1 -28047.245,E2 -28047.245} C_VEL
LIN {X 0,Y 122.566,Z 489.466,A -85,B 0,C 180,E1 -28050.981,E2 -28050.981} C_VEL
LIN {X 0,Y 125.38,Z 486.112,A -85,B 0,C 180,E1 -28052.155,E2 -28052.155} C_VEL
LIN {X 0,Y 126.156,Z 484.284,A -85,B 0,C 180,E1 -28053.533,E2 -28053.533} C_VEL
LIN {X 0,Y 127.151,Z 480.292,A -85,B 0,C 180,E1 -28057.237,E2 -28057.237} C_VEL
LIN {X 0,Y 127.75,Z 477.022,A -85,B 0,C 180,E1 -28060.726,E2 -28060.726} C_VEL
LIN {X 0,Y 128.001,Z 474.62,A -85,B 0,C 180,E1 -28064.065,E2 -28064.065} C_VEL
LIN {X 0,Y 128.071,Z 472.754,A -85,B 0,C 180,E1 -28067.32,E2 -28067.32} C_VEL
LIN {X 0,Y 128.222,Z 471.271,A -85,B 0,C 180,E1 -28070.616,E2 -28070.616} C_VEL
LIN {X 0,Y 128.329,Z 470.385,A -85,B 0,C 180,E1 -28073.711,E2 -28073.711} C_VEL
LIN {X 0,Y 128.426,Z 469.934,A -85,B 0,C 180,E1 -28076.862,E2 -28076.862} C_VEL
LIN {X 0,Y 128.438,Z 470.079,A -85,B 0,C 180,E1 -28079.999,E2 -28079.999} C_VEL
LIN {X 0,Y 128.252,Z 470.981,A -85,B 0,C 180,E1 -28083.141,E2 -28083.141} C_VEL
LIN {X 0,Y 128.099,Z 472.281,A -85,B 0,C 180,E1 -28086.299,E2 -28086.299} C_VEL
LIN {X 0,Y 127.943,Z 474.06,A -85,B 0,C 180,E1 -28089.485,E2 -28089.485} C_VEL
LIN {X 0,Y 127.561,Z 477.813,A -85,B 0,C 180,E1 -28094.354,E2 -28094.354} C_VEL
LIN {X 0,Y 126.714,Z 482.957,A -85,B 0,C 180,E1 -28099.456,E2 -28099.456} C_VEL
LIN {X 0,Y 125.859,Z 487.057,A -85,B 0,C 180,E1 -28103.009,E2 -28103.009} C_VEL
LIN {X 0,Y 125.153,Z 489.166,A -85,B 0,C 180,E1 -28104.488,E2 -28104.488} C_VEL
LIN {X 0,Y 115.264,Z 499.764,A -85,B 0,C 180,E1 -28107.856,E2 -28107.856} C_VEL
LIN {X 0,Y 105.731,Z 508.673,A -85,B 0,C 180,E1 -28111.937,E2 -28111.937} C_VEL
LIN {X 0,Y 96.815,Z 516.176,A -85,B 0,C 180,E1 -28117.01,E2 -28117.01} C_VEL
LIN {X 0,Y 87.59,Z 522.976,A -85,B 0,C 180,E1 -28123.768,E2 -28123.768} C_VEL
LIN {X 0,Y 79.548,Z 528.553,A -85,B 0,C 180,E1 -28132.667,E2 -28132.667} C_VEL
LIN {X 0,Y 74.255,Z 532.132,A -85,B 0,C 180,E1 -28141.755,E2 -28141.755} C_VEL
LIN {X 0,Y 70.742,Z 534.7,A -85,B 0,C 180,E1 -28152.659,E2 -28152.659} C_VEL
LIN {X 0,Y 69.718,Z 536.013,A -85,B 0,C 180,E1 -28164.214,E2 -28164.214} C_VEL
LIN {X 0,Y 69.95,Z 536.193,A -85,B 0,C 180,E1 -28169.999,E2 -28169.999} C_VEL
LIN {X 0,Y 69.719,Z 536.005,A -85,B 0,C 180,E1 -28175.785,E2 -28175.785} C_VEL
LIN {X 0,Y 70.741,Z 534.665,A -85,B 0,C 180,E1 -28187.34,E2 -28187.34} C_VEL
LIN {X 0,Y 74.22,Z 532.07,A -85,B 0,C 180,E1 -28198.259,E2 -28198.259} C_VEL
LIN {X 0,Y 79.889,Z 528.165,A -85,B 0,C 180,E1 -28208.01,E2 -28208.01} C_VEL
LIN {X 0,Y 87.578,Z 522.864,A -85,B 0,C 180,E1 -28216.24,E2 -28216.24} C_VEL
LIN {X 0,Y 96.792,Z 516.026,A -85,B 0,C 180,E1 -28223.007,E2 -28223.007} C_VEL
LIN {X 0,Y 105.564,Z 508.618,A -85,B 0,C 180,E1 -28228.003,E2 -28228.003} C_VEL
LIN {X 0,Y 115.235,Z 499.546,A -85,B 0,C 180,E1 -28232.169,E2 -28232.169} C_VEL
LIN {X 0,Y 125.073,Z 488.953,A -85,B 0,C 180,E1 -28235.52,E2 -28235.52} C_VEL
LIN {X 0,Y 125.501,Z 488.035,A -85,B 0,C 180,E1 -28236.047,E2 -28236.047} C_VEL
LIN {X 0,Y 126.673,Z 482.631,A -85,B 0,C 180,E1 -28240.594,E2 -28240.594} C_VEL
LIN {X 0,Y 127.432,Z 477.631,A -85,B 0,C 180,E1 -28245.631,E2 -28245.631} C_VEL
LIN {X 0,Y 127.827,Z 473.838,A -85,B 0,C 180,E1 -28250.507,E2 -28250.507} C_VEL
LIN {X 0,Y 127.95,Z 472.091,A -85,B 0,C 180,E1 -28253.694,E2 -28253.694} C_VEL
LIN {X 0,Y 128.096,Z 470.784,A -85,B 0,C 180,E1 -28256.855,E2 -28256.855} C_VEL
LIN {X 0,Y 128.324,Z 469.807,A -85,B 0,C 180,E1 -28260.001,E2 -28260.001} C_VEL
LIN {X 0,Y 128.322,Z 469.643,A -85,B 0,C 180,E1 -28263.14,E2 -28263.14} C_VEL
LIN {X 0,Y 128.131,Z 470.502,A -85,B 0,C 180,E1 -28267.67,E2 -28267.67} C_VEL
LIN {X 0,Y 128.115,Z 471.023,A -85,B 0,C 180,E1 -28269.473,E2 -28269.473} C_VEL
LIN {X 0,Y 128.012,Z 472.415,A -85,B 0,C 180,E1 -28272.686,E2 -28272.686} C_VEL
LIN {X 0,Y 127.86,Z 475.11,A -85,B 0,C 180,E1 -28277.132,E2 -28277.132} C_VEL
LIN {X 0,Y 127.355,Z 478.326,A -85,B 0,C 180,E1 -28281.019,E2 -28281.019} C_VEL
LIN {X 0,Y 126.517,Z 482.328,A -85,B 0,C 180,E1 -28285.022,E2 -28285.022} C_VEL
LIN {X 0,Y 125.938,Z 484.376,A -85,B 0,C 180,E1 -28286.762,E2 -28286.762} C_VEL
LIN {X 0,Y 125.309,Z 485.881,A -85,B 0,C 180,E1 -28287.907,E2 -28287.907} C_VEL
LIN {X 0,Y 124.038,Z 487.513,A -85,B 0,C 180,E1 -28288.57,E2 -28288.57} C_VEL
LIN {X 0,Y 115.653,Z 496.302,A -85,B 0,C 180,E1 -28291.707,E2 -28291.707} C_VEL
LIN {X 0,Y 106.21,Z 504.819,A -85,B 0,C 180,E1 -28295.846,E2 -28295.846} C_VEL
LIN {X 0,Y 96.849,Z 512.276,A -85,B 0,C 180,E1 -28301.268,E2 -28301.268} C_VEL
LIN {X 0,Y 89.23,Z 517.694,A -85,B 0,C 180,E1 -28307.114,E2 -28307.114} C_VEL
LIN {X 0,Y 85.513,Z 519.841,A -85,B 0,C 180,E1 -28309.791,E2 -28309.791} C_VEL
LIN {X 0,Y 78.322,Z 522.96,A -85,B 0,C 180,E1 -28314.046,E2 -28314.046} C_VEL
LIN {X 0,Y 72.762,Z 525.071,A -85,B 0,C 180,E1 -28318.051,E2 -28318.051} C_VEL
LIN {X 0,Y 69.47,Z 526.39,A -85,B 0,C 180,E1 -28321.865,E2 -28321.865} C_VEL
LIN {X 0,Y 68.671,Z 526.759,A -85,B 0,C 180,E1 -28323.323,E2 -28323.323} C_VEL
LIN {X 0,Y 65.643,Z 528.354,A -85,B 0,C 180,E1 -28331.265,E2 -28331.265} C_VEL
LIN {X 0,Y 63.329,Z 529.563,A -85,B 0,C 180,E1 -28343.629,E2 -28343.629} C_VEL
LIN {X 0,Y 63.11,Z 529.715,A -85,B 0,C 180,E1 -28350.001,E2 -28350.001} C_VEL
LIN {X 0,Y 64.21,Z 529.136,A -85,B 0,C 180,E1 -28362.646,E2 -28362.646} C_VEL
LIN {X 0,Y 67.667,Z 527.358,A -85,B 0,C 180,E1 -28374.548,E2 -28374.548} C_VEL
LIN {X 0,Y 73.506,Z 524.314,A -85,B 0,C 180,E1 -28385.008,E2 -28385.008} C_VEL
LIN {X 0,Y 81.264,Z 519.925,A -85,B 0,C 180,E1 -28393.779,E2 -28393.779} C_VEL
LIN {X 0,Y 90.542,Z 514.067,A -85,B 0,C 180,E1 -28400.916,E2 -28400.916} C_VEL
LIN {X 0,Y 99.445,Z 507.561,A -85,B 0,C 180,E1 -28406.141,E2 -28406.141} C_VEL
LIN {X 0,Y 109.153,Z 499.573,A -85,B 0,C 180,E1 -28410.37,E2 -28410.37} C_VEL
LIN {X 0,Y 118.958,Z 490.178,A -85,B 0,C 180,E1 -28413.85,E2 -28413.85} C_VEL
LIN {X 0,Y 120.095,Z 488.966,A -85,B 0,C 180,E1 -28414.22,E2 -28414.22} C_VEL
LIN {X 0,Y 121.218,Z 486.681,A -85,B 0,C 180,E1 -28416.055,E2 -28416.055} C_VEL
LIN {X 0,Y 122.325,Z 483.128,A -85,B 0,C 180,E1 -28419.835,E2 -28419.835} C_VEL
LIN {X 0,Y 123.007,Z 480.407,A -85,B 0,C 180,E1 -28423.4,E2 -28423.4} C_VEL
LIN {X 0,Y 123.244,Z 478.465,A -85,B 0,C 180,E1 -28426.814,E2 -28426.814} C_VEL
LIN {X 0,Y 123.516,Z 476.959,A -85,B 0,C 180,E1 -28430.171,E2 -28430.171} C_VEL
LIN {X 0,Y 123.758,Z 475.956,A -85,B 0,C 180,E1 -28433.478,E2 -28433.478} C_VEL
LIN {X 0,Y 123.914,Z 475.465,A -85,B 0,C 180,E1 -28436.748,E2 -28436.748} C_VEL
LIN {X 0,Y 123.921,Z 475.617,A -85,B 0,C 180,E1 -28439.999,E2 -28439.999} C_VEL
LIN {X 0,Y 123.666,Z 476.56,A -85,B 0,C 180,E1 -28443.257,E2 -28443.257} C_VEL
LIN {X 0,Y 123.406,Z 477.917,A -85,B 0,C 180,E1 -28446.54,E2 -28446.54} C_VEL
LIN {X 0,Y 122.816,Z 481.132,A -85,B 0,C 180,E1 -28451.72,E2 -28451.72} C_VEL
LIN {X 0,Y 122.234,Z 483.844,A -85,B 0,C 180,E1 -28454.994,E2 -28454.994} C_VEL
LIN {X 0,Y 121.193,Z 487.987,A -85,B 0,C 180,E1 -28459.229,E2 -28459.229} C_VEL
LIN {X 0,Y 120.612,Z 490.07,A -85,B 0,C 180,E1 -28461.199,E2 -28461.199} C_VEL
LIN {X 0,Y 120.143,Z 491.159,A -85,B 0,C 180,E1 -28462.045,E2 -28462.045} C_VEL
LIN {X 0,Y 110.631,Z 500.767,A -85,B 0,C 180,E1 -28465.141,E2 -28465.141} C_VEL
LIN {X 0,Y 101.249,Z 509.016,A -85,B 0,C 180,E1 -28468.905,E2 -28468.905} C_VEL
LIN {X 0,Y 92.656,Z 515.821,A -85,B 0,C 180,E1 -28473.449,E2 -28473.449} C_VEL
LIN {X 0,Y 82.785,Z 522.625,A -85,B 0,C 180,E1 -28480.176,E2 -28480.176} C_VEL
LIN {X 0,Y 74.452,Z 527.902,A -85,B 0,C 180,E1 -28488.64,E2 -28488.64} C_VEL
LIN {X 0,Y 68.006,Z 531.783,A -85,B 0,C 180,E1 -28498.887,E2 -28498.887} C_VEL
LIN {X 0,Y 63.946,Z 534.353,A -85,B 0,C 180,E1 -28510.748,E2 -28510.748} C_VEL
LIN {X 0,Y 62.615,Z 535.666,A -85,B 0,C 180,E1 -28523.555,E2 -28523.555} C_VEL
LIN {X 0,Y 62.844,Z 535.847,A -85,B 0,C 180,E1 -28529.999,E2 -28529.999} C_VEL
LIN {X 0,Y 62.616,Z 535.657,A -85,B 0,C 180,E1 -28536.444,E2 -28536.444} C_VEL
LIN {X 0,Y 63.943,Z 534.317,A -85,B 0,C 180,E1 -28549.252,E2 -28549.252} C_VEL
LIN {X 0,Y 67.966,Z 531.719,A -85,B 0,C 180,E1 -28561.132,E2 -28561.132} C_VEL
LIN {X 0,Y 74.365,Z 527.814,A -85,B 0,C 180,E1 -28571.418,E2 -28571.418} C_VEL
LIN {X 0,Y 82.775,Z 522.512,A -85,B 0,C 180,E1 -28579.831,E2 -28579.831} C_VEL
LIN {X 0,Y 92.627,Z 515.667,A -85,B 0,C 180,E1 -28586.576,E2 -28586.576} C_VEL
LIN {X 0,Y 102.079,Z 508.14,A -85,B 0,C 180,E1 -28591.493,E2 -28591.493} C_VEL
LIN {X 0,Y 112.074,Z 499.175,A -85,B 0,C 180,E1 -28595.406,E2 -28595.406} C_VEL
LIN {X 0,Y 120.048,Z 490.974,A -85,B 0,C 180,E1 -28597.952,E2 -28597.952} C_VEL
LIN {X 0,Y 120.786,Z 489.041,A -85,B 0,C 180,E1 -28599.568,E2 -28599.568} C_VEL
LIN {X 0,Y 121.744,Z 485.267,A -85,B 0,C 180,E1 -28603.224,E2 -28603.224} C_VEL
LIN {X 0,Y 122.539,Z 481.791,A -85,B 0,C 180,E1 -28607.163,E2 -28607.163} C_VEL
LIN {X 0,Y 122.94,Z 479.62,A -85,B 0,C 180,E1 -28610.126,E2 -28610.126} C_VEL
LIN {X 0,Y 123.271,Z 477.726,A -85,B 0,C 180,E1 -28613.453,E2 -28613.453} C_VEL
LIN {X 0,Y 123.516,Z 476.369,A -85,B 0,C 180,E1 -28616.739,E2 -28616.739} C_VEL
LIN {X 0,Y 123.809,Z 475.365,A -85,B 0,C 180,E1 -28620.001,E2 -28620.001} C_VEL
LIN {X 0,Y 123.818,Z 475.187,A -85,B 0,C 180,E1 -28623.254,E2 -28623.254} C_VEL
LIN {X 0,Y 123.535,Z 476.018,A -85,B 0,C 180,E1 -28627.59,E2 -28627.59} C_VEL
